LIN {X 0.241,Y -599.129,Z 1375.125,A 0.000,B 0.000,C 90.000,E1 58.408} C_DIS
LIN {X 0.169,Y -600.635,Z 1375.116,A 0.000,B 0.000,C 90.000,E1 56.834} C_DIS
LIN {X -0.271,Y -601.408,Z 1375.111,A 0.000,B 0.000,C 90.000,E1 56.087} C_DIS
LIN {X 0.294,Y -603.031,Z 1375.101,A 0.000,B 0.000,C 90.000,E1 54.196} C_DIS
LIN {X -0.072,Y -604.729,Z 1375.091,A 0.000,B 0.000,C 90.000,E1 52.396} C_DIS
LIN {X -0.082,Y -605.645,Z 1375.084,A 0.000,B 0.000,C 90.000,E1 51.090} C_DIS
LIN {X 0.038,Y -606.172,Z 1375.078,A 0.000,B 0.000,C 90.000,E1 50.033} C_DIS
LIN {X -0.227,Y -606.705,Z 1375.072,A 0.000,B 0.000,C 90.000,E1 49.013} C_DIS
LIN {X -0.356,Y -607.003,Z 1375.068,A 0.000,B 0.000,C 90.000,E1 48.243} C_DIS
LIN {X -0.003,Y -607.306,Z 1375.061,A 0.000,B 0.000,C 90.000,E1 46.905} C_DIS
LIN {X 0.356,Y -607.367,Z 1375.053,A 0.000,B 0.000,C 90.000,E1 45.567} C_DIS
LIN {X -0.205,Y -607.319,Z 1375.049,A 0.000,B 0.000,C 90.000,E1 44.838} C_DIS
LIN {X -0.286,Y -606.975,Z 1375.042,A 0.000,B 0.000,C 90.000,E1 43.542} C_DIS
LIN {X 0.058,Y -606.352,Z 1375.035,A 0.000,B 0.000,C 90.000,E1 42.204} C_DIS
LIN {X -0.017,Y -605.691,Z 1375.027,A 0.000,B 0.000,C 90.000,E1 40.906} C_DIS
LIN {X 0.357,Y -604.817,Z 1375.020,A 0.000,B 0.000,C 90.000,E1 39.564} C_DIS
LIN {X -0.137,Y -603.773,Z 1375.013,A 0.000,B 0.000,C 90.000,E1 38.302} C_DIS
LIN {X -0.179,Y -602.457,Z 1375.005,A 0.000,B 0.000,C 90.000,E1 36.996} C_DIS
LIN {X 0.222,Y -601.485,Z 1375.001,A 0.000,B 0.000,C 90.000,E1 36.171} C_DIS
LIN {X -0.113,Y -599.795,Z 1374.995,A 0.000,B 0.000,C 90.000,E1 35.152} C_DIS
LIN {X -0.215,Y -599.352,Z 1374.994,A 0.000,B 0.000,C 90.000,E1 34.898} C_DIS
LIN {X -0.198,Y -596.501,Z 1374.986,A 0.000,B 0.000,C 90.000,E1 33.579} C_DIS
LIN {X 0.149,Y -594.609,Z 1374.982,A 0.000,B 0.000,C 90.000,E1 32.752} C_DIS
LIN {X -0.345,Y -592.452,Z 1374.978,A 0.000,B 0.000,C 90.000,E1 32.005} C_DIS
LIN {X -0.050,Y -590.090,Z 1374.973,A 0.000,B 0.000,C 90.000,E1 31.180} C_DIS
LIN {X -0.205,Y -586.275,Z 1374.967,A 0.000,B 0.000,C 90.000,E1 30.129} C_DIS
LIN {X 0.229,Y -583.094,Z 1374.963,A 0.000,B 0.000,C 90.000,E1 29.283} C_DIS
LIN {X 0.119,Y -579.414,Z 1374.958,A 0.000,B 0.000,C 90.000,E1 28.487} C_DIS
LIN {X -0.235,Y -576.095,Z 1374.955,A 0.000,B 0.000,C 90.000,E1 27.847} C_DIS
LIN {X 0.082,Y -571.788,Z 1374.950,A 0.000,B 0.000,C 90.000,E1 27.001} C_DIS
LIN {X 0.091,Y -567.040,Z 1374.946,A 0.000,B 0.000,C 90.000,E1 26.181} C_DIS
LIN {X -0.022,Y -563.676,Z 1374.943,A 0.000,B 0.000,C 90.000,E1 25.643} C_DIS
LIN {X -0.098,Y -558.415,Z 1374.938,A 0.000,B 0.000,C 90.000,E1 24.823} C_DIS
LIN {X 0.162,Y -551.372,Z 1374.932,A 0.000,B 0.000,C 90.000,E1 23.823} C_DIS
LIN {X 0.076,Y -545.974,Z 1374.929,A 0.000,B 0.000,C 90.000,E1 23.131} C_DIS
LIN {X -0.265,Y -540.164,Z 1374.925,A 0.000,B 0.000,C 90.000,E1 22.461} C_DIS
LIN {X -0.093,Y -532.857,Z 1374.920,A 0.000,B 0.000,C 90.000,E1 21.589} C_DIS
LIN {X -0.184,Y -522.480,Z 1374.914,A 0.000,B 0.000,C 90.000,E1 20.482} C_DIS
LIN {X -0.189,Y -513.235,Z 1374.908,A 0.000,B 0.000,C 90.000,E1 19.504} C_DIS
LIN {X -0.122,Y -502.645,Z 1374.902,A 0.000,B 0.000,C 90.000,E1 18.417} C_DIS
LIN {X 0.112,Y -491.666,Z 1374.896,A 0.000,B 0.000,C 90.000,E1 17.275} C_DIS
LIN {X -0.037,Y -476.636,Z 1374.888,A 0.000,B 0.000,C 90.000,E1 15.788} C_DIS
LIN {X 0.103,Y -466.836,Z 1374.882,A 0.000,B 0.000,C 90.000,E1 14.773} C_DIS
LIN {X 0.103,Y -454.064,Z 1374.875,A 0.000,B 0.000,C 90.000,E1 13.480} C_DIS
LIN {X -0.045,Y -437.083,Z 1374.865,A 0.000,B 0.000,C 90.000,E1 11.715} C_DIS
LIN {X -0.036,Y -421.953,Z 1374.856,A 0.000,B 0.000,C 90.000,E1 10.018} C_DIS
LIN {X 0.137,Y -410.842,Z 1374.848,A 0.000,B 0.000,C 90.000,E1 8.690} C_DIS
LIN {X 0.106,Y -402.395,Z 1374.843,A 0.000,B 0.000,C 90.000,E1 7.701} C_DIS
LIN {X -0.087,Y -396.749,Z 1374.839,A 0.000,B 0.000,C 90.000,E1 7.068} C_DIS
LIN {X -0.005,Y -393.047,Z 1374.836,A 0.000,B 0.000,C 90.000,E1 6.549} C_DIS
LIN {X -0.180,Y -391.673,Z 1374.835,A 0.000,B 0.000,C 90.000,E1 6.315} C_DIS
LIN {X 0.172,Y -391.657,Z 1374.835,A 0.000,B 0.000,C 90.000,E1 6.258} C_DIS
LIN {X 0.125,Y -394.271,Z 1374.833,A 0.000,B 0.000,C 90.000,E1 5.910} C_DIS
LIN {X 0.119,Y -398.146,Z 1374.831,A 0.000,B 0.000,C 90.000,E1 5.568} C_DIS
LIN {X 0.042,Y -406.599,Z 1374.828,A 0.000,B 0.000,C 90.000,E1 4.935} C_DIS
LIN {X -0.167,Y -411.326,Z 1374.825,A 0.000,B 0.000,C 90.000,E1 4.588} C_DIS
LIN {X -0.196,Y -415.671,Z 1374.823,A 0.000,B 0.000,C 90.000,E1 4.188} C_DIS
LIN {X 0.010,Y -419.888,Z 1374.821,A 0.000,B 0.000,C 90.000,E1 3.726} C_DIS
LIN {X 0.095,Y -424.949,Z 1374.818,A 0.000,B 0.000,C 90.000,E1 3.154} C_DIS
LIN {X -0.129,Y -430.292,Z 1374.814,A 0.000,B 0.000,C 90.000,E1 2.522} C_DIS
LIN {X -0.086,Y -436.249,Z 1374.810,A 0.000,B 0.000,C 90.000,E1 1.718} C_DIS
LIN {X 0.170,Y -442.273,Z 1374.805,A 0.000,B 0.000,C 90.000,E1 0.859} C_DIS
LIN {X 0.000,Y -448.347,Z 1374.800,A 0.000,B 0.000,C 90.000,E1 360.000} C_DIS
LIN {X 0.033,Y -453.864,Z 1374.795,A 0.000,B 0.000,C 90.000,E1 359.141} C_DIS
LIN {X 0.020,Y -458.743,Z 1374.791,A 0.000,B 0.000,C 90.000,E1 358.339} C_DIS
LIN {X -0.035,Y -462.399,Z 1374.787,A 0.000,B 0.000,C 90.000,E1 357.707} C_DIS
LIN {X 0.164,Y -467.432,Z 1374.782,A 0.000,B 0.000,C 90.000,E1 356.731} C_DIS
LIN {X 0.153,Y -470.561,Z 1374.778,A 0.000,B 0.000,C 90.000,E1 356.102} C_DIS
LIN {X -0.152,Y -474.160,Z 1374.774,A 0.000,B 0.000,C 90.000,E1 355.355} C_DIS
LIN {X 0.222,Y -478.076,Z 1374.769,A 0.000,B 0.000,C 90.000,E1 354.375} C_DIS
LIN {X -0.150,Y -480.507,Z 1374.766,A 0.000,B 0.000,C 90.000,E1 353.799} C_DIS
LIN {X -0.181,Y -483.879,Z 1374.760,A 0.000,B 0.000,C 90.000,E1 352.875} C_DIS
LIN {X -0.040,Y -485.914,Z 1374.757,A 0.000,B 0.000,C 90.000,E1 352.243} C_DIS
LIN {X -0.013,Y -488.702,Z 1374.752,A 0.000,B 0.000,C 90.000,E1 351.319} C_DIS
LIN {X -0.250,Y -490.361,Z 1374.748,A 0.000,B 0.000,C 90.000,E1 350.735} C_DIS
LIN {X -0.196,Y -493.358,Z 1374.742,A 0.000,B 0.000,C 90.000,E1 349.511} C_DIS
LIN {X 0.092,Y -494.730,Z 1374.738,A 0.000,B 0.000,C 90.000,E1 348.870} C_DIS
LIN {X -0.002,Y -495.337,Z 1374.737,A 0.000,B 0.000,C 90.000,E1 348.578} C_DIS
LIN {X -0.094,Y -495.813,Z 1374.735,A 0.000,B 0.000,C 90.000,E1 348.285} C_DIS
LIN {X -0.184,Y -496.075,Z 1374.733,A 0.000,B 0.000,C 90.000,E1 347.993} C_DIS
LIN {X 0.212,Y -496.110,Z 1374.732,A 0.000,B 0.000,C 90.000,E1 347.645} C_DIS
LIN {X 0.123,Y -495.824,Z 1374.730,A 0.000,B 0.000,C 90.000,E1 347.353} C_DIS
LIN {X 0.034,Y -494.778,Z 1374.728,A 0.000,B 0.000,C 90.000,E1 347.061} C_DIS
LIN {X -0.129,Y -493.185,Z 1374.727,A 0.000,B 0.000,C 90.000,E1 346.937} C_DIS
LIN {X 0.101,Y -455.532,Z 1374.721,A 0.000,B 0.000,C 90.000,E1 345.825} C_DIS
LIN {X 0.169,Y -423.917,Z 1374.715,A 0.000,B 0.000,C 90.000,E1 344.755} C_DIS
LIN {X 0.093,Y -395.987,Z 1374.709,A 0.000,B 0.000,C 90.000,E1 343.685} C_DIS
LIN {X 0.175,Y -371.706,Z 1374.703,A 0.000,B 0.000,C 90.000,E1 342.598} C_DIS
LIN {X 0.086,Y -360.270,Z 1374.700,A 0.000,B 0.000,C 90.000,E1 342.054} C_DIS
LIN {X 0.052,Y -360.184,Z 1374.700,A 0.000,B 0.000,C 90.000,E1 342.054} C_DIS
LIN {X -0.028,Y -361.934,Z 1374.683,A 0.000,B 0.000,C 90.000,E1 338.954} C_DIS
LIN {X -0.170,Y -366.154,Z 1374.642,A 0.000,B 0.000,C 90.000,E1 331.513} C_DIS
LIN {X 0.050,Y -371.141,Z 1374.605,A 0.000,B 0.000,C 90.000,E1 324.815} C_DIS
LIN {X -0.178,Y -371.570,Z 1374.603,A 0.000,B 0.000,C 90.000,E1 324.482} C_DIS
LIN {X 0.098,Y -372.300,Z 1374.596,A 0.000,B 0.000,C 90.000,E1 323.336} C_DIS
LIN {X 0.155,Y -378.074,Z 1374.564,A 0.000,B 0.000,C 90.000,E1 317.472} C_DIS
LIN {X 0.177,Y -384.183,Z 1374.530,A 0.000,B 0.000,C 90.000,E1 311.310} C_DIS
LIN {X -0.070,Y -384.685,Z 1374.528,A 0.000,B 0.000,C 90.000,E1 310.987} C_DIS
LIN {X -0.170,Y -385.795,Z 1374.520,A 0.000,B 0.000,C 90.000,E1 309.564} C_DIS
LIN {X -0.011,Y -391.319,Z 1374.492,A 0.000,B 0.000,C 90.000,E1 304.532} C_DIS
LIN {X 0.135,Y -397.031,Z 1374.458,A 0.000,B 0.000,C 90.000,E1 298.487} C_DIS
LIN {X -0.084,Y -401.405,Z 1374.427,A 0.000,B 0.000,C 90.000,E1 292.898} C_DIS
LIN {X 0.151,Y -401.668,Z 1374.425,A 0.000,B 0.000,C 90.000,E1 292.514} C_DIS
LIN {X -0.104,Y -404.762,Z 1374.394,A 0.000,B 0.000,C 90.000,E1 286.968} C_DIS
LIN {X -0.209,Y -406.158,Z 1374.363,A 0.000,B 0.000,C 90.000,E1 281.422} C_DIS
LIN {X -0.105,Y -405.652,Z 1374.333,A 0.000,B 0.000,C 90.000,E1 275.853} C_DIS
LIN {X -0.033,Y -403.559,Z 1374.305,A 0.000,B 0.000,C 90.000,E1 270.974} C_DIS
LIN {X -0.098,Y -403.120,Z 1374.302,A 0.000,B 0.000,C 90.000,E1 270.286} C_DIS
LIN {X 0.131,Y -399.041,Z 1374.272,A 0.000,B 0.000,C 90.000,E1 265.008} C_DIS
LIN {X 0.072,Y -398.696,Z 1374.271,A 0.000,B 0.000,C 90.000,E1 264.666} C_DIS
LIN {X -0.046,Y -393.247,Z 1374.243,A 0.000,B 0.000,C 90.000,E1 259.746} C_DIS
LIN {X -0.085,Y -392.976,Z 1374.241,A 0.000,B 0.000,C 90.000,E1 259.398} C_DIS
LIN {X -0.126,Y -392.577,Z 1374.239,A 0.000,B 0.000,C 90.000,E1 259.050} C_DIS
LIN {X 0.033,Y -386.186,Z 1374.213,A 0.000,B 0.000,C 90.000,E1 254.393} C_DIS
LIN {X -0.004,Y -385.081,Z 1374.207,A 0.000,B 0.000,C 90.000,E1 253.323} C_DIS
LIN {X 0.100,Y -378.210,Z 1374.183,A 0.000,B 0.000,C 90.000,E1 248.975} C_DIS
LIN {X -0.044,Y -375.993,Z 1374.173,A 0.000,B 0.000,C 90.000,E1 247.177} C_DIS
LIN {X 0.067,Y -369.190,Z 1374.151,A 0.000,B 0.000,C 90.000,E1 243.127} C_DIS
LIN {X -0.025,Y -366.331,Z 1374.139,A 0.000,B 0.000,C 90.000,E1 240.923} C_DIS
LIN {X 0.133,Y -358.937,Z 1374.114,A 0.000,B 0.000,C 90.000,E1 236.421} C_DIS
LIN {X -0.078,Y -356.112,Z 1374.101,A 0.000,B 0.000,C 90.000,E1 234.196} C_DIS
LIN {X 0.018,Y -349.041,Z 1374.076,A 0.000,B 0.000,C 90.000,E1 229.622} C_DIS
LIN {X -0.016,Y -345.986,Z 1374.061,A 0.000,B 0.000,C 90.000,E1 226.944} C_DIS
LIN {X -0.043,Y -339.190,Z 1374.033,A 0.000,B 0.000,C 90.000,E1 221.919} C_DIS
LIN {X 0.045,Y -337.008,Z 1374.020,A 0.000,B 0.000,C 90.000,E1 219.564} C_DIS
LIN {X 0.021,Y -336.054,Z 1374.016,A 0.000,B 0.000,C 90.000,E1 218.785} C_DIS
LIN {X -0.099,Y -330.416,Z 1373.985,A 0.000,B 0.000,C 90.000,E1 213.293} C_DIS
LIN {X 0.206,Y -329.135,Z 1373.974,A 0.000,B 0.000,C 90.000,E1 211.258} C_DIS
LIN {X 0.083,Y -324.407,Z 1373.938,A 0.000,B 0.000,C 90.000,E1 204.899} C_DIS
LIN {X 0.071,Y -323.717,Z 1373.927,A 0.000,B 0.000,C 90.000,E1 202.898} C_DIS
LIN {X -0.060,Y -322.264,Z 1373.914,A 0.000,B 0.000,C 90.000,E1 200.556} C_DIS
LIN {X -0.078,Y -322.271,Z 1373.914,A 0.000,B 0.000,C 90.000,E1 200.556} C_DIS
LIN {X 0.093,Y -344.041,Z 1373.907,A 0.000,B 0.000,C 90.000,E1 199.214} C_DIS
LIN {X 0.091,Y -367.098,Z 1373.900,A 0.000,B 0.000,C 90.000,E1 198.000} C_DIS
LIN {X -0.130,Y -393.883,Z 1373.893,A 0.000,B 0.000,C 90.000,E1 196.804} C_DIS
LIN {X -0.144,Y -422.596,Z 1373.887,A 0.000,B 0.000,C 90.000,E1 195.662} C_DIS
LIN {X -0.056,Y -440.653,Z 1373.883,A 0.000,B 0.000,C 90.000,E1 195.009} C_DIS
LIN {X -0.145,Y -443.464,Z 1373.883,A 0.000,B 0.000,C 90.000,E1 194.898} C_DIS
LIN {X 0.077,Y -444.638,Z 1373.882,A 0.000,B 0.000,C 90.000,E1 194.717} C_DIS
LIN {X 0.212,Y -445.410,Z 1373.881,A 0.000,B 0.000,C 90.000,E1 194.537} C_DIS
LIN {X -0.084,Y -445.964,Z 1373.880,A 0.000,B 0.000,C 90.000,E1 194.411} C_DIS
LIN {X 0.082,Y -446.725,Z 1373.878,A 0.000,B 0.000,C 90.000,E1 194.064} C_DIS
LIN {X -0.182,Y -447.189,Z 1373.876,A 0.000,B 0.000,C 90.000,E1 193.772} C_DIS
LIN {X 0.098,Y -447.488,Z 1373.875,A 0.000,B 0.000,C 90.000,E1 193.411} C_DIS
LIN {X 0.044,Y -447.972,Z 1373.867,A 0.000,B 0.000,C 90.000,E1 192.119} C_DIS
LIN {X -0.092,Y -448.344,Z 1373.860,A 0.000,B 0.000,C 90.000,E1 190.838} C_DIS
LIN {X -0.031,Y -448.520,Z 1373.851,A 0.000,B 0.000,C 90.000,E1 189.208} C_DIS
LIN {X -0.108,Y -448.510,Z 1373.839,A 0.000,B 0.000,C 90.000,E1 186.947} C_DIS
LIN {X 0.087,Y -448.469,Z 1373.831,A 0.000,B 0.000,C 90.000,E1 185.625} C_DIS
LIN {X 0.145,Y -448.331,Z 1373.826,A 0.000,B 0.000,C 90.000,E1 184.645} C_DIS
LIN {X -0.140,Y -447.861,Z 1373.819,A 0.000,B 0.000,C 90.000,E1 183.383} C_DIS
LIN {X 0.176,Y -447.483,Z 1373.815,A 0.000,B 0.000,C 90.000,E1 182.694} C_DIS
LIN {X 0.181,Y -446.518,Z 1373.810,A 0.000,B 0.000,C 90.000,E1 181.718} C_DIS
LIN {X 0.020,Y -445.840,Z 1373.806,A 0.000,B 0.000,C 90.000,E1 181.088} C_DIS
LIN {X -0.143,Y -445.025,Z 1373.802,A 0.000,B 0.000,C 90.000,E1 180.458} C_DIS
LIN {X -0.176,Y -443.449,Z 1373.797,A 0.000,B 0.000,C 90.000,E1 179.484} C_DIS
LIN {X 0.086,Y -442.211,Z 1373.793,A 0.000,B 0.000,C 90.000,E1 178.797} C_DIS
LIN {X 0.029,Y -439.643,Z 1373.788,A 0.000,B 0.000,C 90.000,E1 177.822} C_DIS
LIN {X -0.181,Y -437.692,Z 1373.784,A 0.000,B 0.000,C 90.000,E1 177.192} C_DIS
LIN {X 0.053,Y -435.361,Z 1373.781,A 0.000,B 0.000,C 90.000,E1 176.502} C_DIS
LIN {X 0.192,Y -433.388,Z 1373.778,A 0.000,B 0.000,C 90.000,E1 175.988} C_DIS
LIN {X -0.047,Y -430.543,Z 1373.774,A 0.000,B 0.000,C 90.000,E1 175.355} C_DIS
LIN {X 0.216,Y -425.262,Z 1373.769,A 0.000,B 0.000,C 90.000,E1 174.318} C_DIS
LIN {X -0.006,Y -418.909,Z 1373.763,A 0.000,B 0.000,C 90.000,E1 173.337} C_DIS
LIN {X 0.112,Y -412.069,Z 1373.757,A 0.000,B 0.000,C 90.000,E1 172.299} C_DIS
LIN {X 0.155,Y -398.379,Z 1373.746,A 0.000,B 0.000,C 90.000,E1 170.218} C_DIS
LIN {X 0.055,Y -387.770,Z 1373.736,A 0.000,B 0.000,C 90.000,E1 168.465} C_DIS
LIN {X -0.070,Y -383.203,Z 1373.731,A 0.000,B 0.000,C 90.000,E1 167.589} C_DIS
LIN {X 0.044,Y -380.586,Z 1373.727,A 0.000,B 0.000,C 90.000,E1 166.881} C_DIS
LIN {X 0.042,Y -380.052,Z 1373.726,A 0.000,B 0.000,C 90.000,E1 166.700} C_DIS
LIN {X -0.148,Y -380.021,Z 1373.724,A 0.000,B 0.000,C 90.000,E1 166.353} C_DIS
LIN {X -0.169,Y -380.030,Z 1373.724,A 0.000,B 0.000,C 90.000,E1 166.353} C_DIS
LIN {X -0.062,Y -381.121,Z 1373.723,A 0.000,B 0.000,C 90.000,E1 166.117} C_DIS
LIN {X -0.050,Y -382.411,Z 1373.721,A 0.000,B 0.000,C 90.000,E1 165.811} C_DIS
LIN {X 0.017,Y -387.298,Z 1373.718,A 0.000,B 0.000,C 90.000,E1 165.172} C_DIS
LIN {X -0.039,Y -393.789,Z 1373.714,A 0.000,B 0.000,C 90.000,E1 164.448} C_DIS
LIN {X -0.086,Y -400.930,Z 1373.710,A 0.000,B 0.000,C 90.000,E1 163.740} C_DIS
LIN {X 0.039,Y -416.462,Z 1373.702,A 0.000,B 0.000,C 90.000,E1 162.308} C_DIS
LIN {X 0.224,Y -441.867,Z 1373.690,A 0.000,B 0.000,C 90.000,E1 160.242} C_DIS
LIN {X -0.082,Y -454.491,Z 1373.685,A 0.000,B 0.000,C 90.000,E1 159.316} C_DIS
LIN {X -0.007,Y -460.608,Z 1373.682,A 0.000,B 0.000,C 90.000,E1 158.827} C_DIS
LIN {X -0.071,Y -468.194,Z 1373.679,A 0.000,B 0.000,C 90.000,E1 158.209} C_DIS
LIN {X 0.167,Y -475.655,Z 1373.675,A 0.000,B 0.000,C 90.000,E1 157.539} C_DIS
LIN {X -0.219,Y -484.360,Z 1373.671,A 0.000,B 0.000,C 90.000,E1 156.794} C_DIS
LIN {X -0.096,Y -492.955,Z 1373.667,A 0.000,B 0.000,C 90.000,E1 155.973} C_DIS
LIN {X -0.149,Y -501.060,Z 1373.662,A 0.000,B 0.000,C 90.000,E1 155.153} C_DIS
LIN {X -0.035,Y -505.036,Z 1373.660,A 0.000,B 0.000,C 90.000,E1 154.717} C_DIS
LIN {X 0.113,Y -511.378,Z 1373.656,A 0.000,B 0.000,C 90.000,E1 153.973} C_DIS
LIN {X -0.074,Y -517.595,Z 1373.651,A 0.000,B 0.000,C 90.000,E1 153.256} C_DIS
LIN {X 0.254,Y -523.274,Z 1373.647,A 0.000,B 0.000,C 90.000,E1 152.487} C_DIS
LIN {X -0.227,Y -526.484,Z 1373.645,A 0.000,B 0.000,C 90.000,E1 152.103} C_DIS
LIN {X -0.133,Y -530.224,Z 1373.642,A 0.000,B 0.000,C 90.000,E1 151.513} C_DIS
LIN {X -0.156,Y -534.214,Z 1373.638,A 0.000,B 0.000,C 90.000,E1 150.795} C_DIS
LIN {X -0.002,Y -536.963,Z 1373.635,A 0.000,B 0.000,C 90.000,E1 150.205} C_DIS
LIN {X 0.165,Y -540.360,Z 1373.630,A 0.000,B 0.000,C 90.000,E1 149.331} C_DIS
LIN {X -0.103,Y -542.398,Z 1373.627,A 0.000,B 0.000,C 90.000,E1 148.791} C_DIS
LIN {X 0.106,Y -544.198,Z 1373.623,A 0.000,B 0.000,C 90.000,E1 148.201} C_DIS
LIN {X -0.107,Y -546.401,Z 1373.619,A 0.000,B 0.000,C 90.000,E1 147.375} C_DIS
LIN {X 0.125,Y -547.666,Z 1373.616,A 0.000,B 0.000,C 90.000,E1 146.786} C_DIS
LIN {X -0.052,Y -549.270,Z 1373.611,A 0.000,B 0.000,C 90.000,E1 145.960} C_DIS
LIN {X 0.157,Y -551.091,Z 1373.605,A 0.000,B 0.000,C 90.000,E1 144.815} C_DIS
LIN {X 0.014,Y -552.233,Z 1373.600,A 0.000,B 0.000,C 90.000,E1 143.989} C_DIS
LIN {X 0.273,Y -553.255,Z 1373.594,A 0.000,B 0.000,C 90.000,E1 142.844} C_DIS
LIN {X 0.181,Y -554.267,Z 1373.586,A 0.000,B 0.000,C 90.000,E1 141.457} C_DIS
LIN {X 0.033,Y -555.029,Z 1373.580,A 0.000,B 0.000,C 90.000,E1 140.356} C_DIS
LIN {X 0.320,Y -555.830,Z 1373.572,A 0.000,B 0.000,C 90.000,E1 138.933} C_DIS
LIN {X 0.200,Y -556.587,Z 1373.564,A 0.000,B 0.000,C 90.000,E1 137.553} C_DIS
LIN {X -0.318,Y -557.169,Z 1373.557,A 0.000,B 0.000,C 90.000,E1 136.215} C_DIS
LIN {X 0.014,Y -557.779,Z 1373.547,A 0.000,B 0.000,C 90.000,E1 134.514} C_DIS
LIN {X -0.099,Y -558.296,Z 1373.540,A 0.000,B 0.000,C 90.000,E1 133.137} C_DIS
LIN {X -0.180,Y -558.783,Z 1373.532,A 0.000,B 0.000,C 90.000,E1 131.757} C_DIS
LIN {X 0.011,Y -559.850,Z 1373.520,A 0.000,B 0.000,C 90.000,E1 129.519} C_DIS
LIN {X -0.046,Y -560.355,Z 1373.517,A 0.000,B 0.000,C 90.000,E1 129.116} C_DIS
LIN {X -0.082,Y -561.346,Z 1373.515,A 0.000,B 0.000,C 90.000,E1 128.705} C_DIS
LIN {X 0.082,Y -561.467,Z 1373.515,A 0.000,B 0.000,C 90.000,E1 128.588} C_DIS
LIN {X 0.040,Y -561.486,Z 1373.514,A 0.000,B 0.000,C 90.000,E1 128.588} C_DIS
LIN {X -0.088,Y -562.514,Z 1373.514,A 0.000,B 0.000,C 90.000,E1 128.463} C_DIS
LIN {X -0.117,Y -564.716,Z 1373.513,A 0.000,B 0.000,C 90.000,E1 128.338} C_DIS
LIN {X -0.017,Y -569.709,Z 1373.512,A 0.000,B 0.000,C 90.000,E1 128.177} C_DIS
LIN {X 0.216,Y -572.168,Z 1373.512,A 0.000,B 0.000,C 90.000,E1 128.096} C_DIS
LIN {X -0.017,Y -578.338,Z 1373.511,A 0.000,B 0.000,C 90.000,E1 127.935} C_DIS
LIN {X 0.144,Y -581.541,Z 1373.510,A 0.000,B 0.000,C 90.000,E1 127.810} C_DIS
LIN {X -0.252,Y -584.383,Z 1373.510,A 0.000,B 0.000,C 90.000,E1 127.729} C_DIS
LIN {X -0.065,Y -587.357,Z 1373.509,A 0.000,B 0.000,C 90.000,E1 127.569} C_DIS
LIN {X 0.067,Y -590.363,Z 1373.508,A 0.000,B 0.000,C 90.000,E1 127.397} C_DIS
LIN {X -0.042,Y -593.196,Z 1373.507,A 0.000,B 0.000,C 90.000,E1 127.237} C_DIS
LIN {X -0.077,Y -598.802,Z 1373.505,A 0.000,B 0.000,C 90.000,E1 126.870} C_DIS
LIN {X -0.088,Y -604.276,Z 1373.503,A 0.000,B 0.000,C 90.000,E1 126.457} C_DIS
LIN {X 0.234,Y -608.428,Z 1373.501,A 0.000,B 0.000,C 90.000,E1 126.091} C_DIS
LIN {X 0.068,Y -614.929,Z 1373.497,A 0.000,B 0.000,C 90.000,E1 125.518} C_DIS
LIN {X 0.120,Y -621.206,Z 1373.494,A 0.000,B 0.000,C 90.000,E1 124.898} C_DIS
LIN {X 0.012,Y -626.001,Z 1373.491,A 0.000,B 0.000,C 90.000,E1 124.405} C_DIS
LIN {X -0.152,Y -630.526,Z 1373.488,A 0.000,B 0.000,C 90.000,E1 123.913} C_DIS
LIN {X -0.295,Y -636.832,Z 1373.484,A 0.000,B 0.000,C 90.000,E1 123.166} C_DIS
LIN {X 0.142,Y -641.613,Z 1373.481,A 0.000,B 0.000,C 90.000,E1 122.498} C_DIS
LIN {X 0.082,Y -646.017,Z 1373.477,A 0.000,B 0.000,C 90.000,E1 121.878} C_DIS
LIN {X 0.013,Y -649.279,Z 1373.474,A 0.000,B 0.000,C 90.000,E1 121.386} C_DIS
LIN {X 0.183,Y -652.248,Z 1373.472,A 0.000,B 0.000,C 90.000,E1 120.875} C_DIS
LIN {X 0.332,Y -655.444,Z 1373.468,A 0.000,B 0.000,C 90.000,E1 120.256} C_DIS
LIN {X 0.093,Y -658.704,Z 1373.464,A 0.000,B 0.000,C 90.000,E1 119.539} C_DIS
LIN {X -0.113,Y -661.218,Z 1373.460,A 0.000,B 0.000,C 90.000,E1 118.821} C_DIS
LIN {X -0.294,Y -662.986,Z 1373.456,A 0.000,B 0.000,C 90.000,E1 118.103} C_DIS
LIN {X -0.013,Y -663.616,Z 1373.453,A 0.000,B 0.000,C 90.000,E1 117.590} C_DIS
LIN {X -0.172,Y -663.947,Z 1373.449,A 0.000,B 0.000,C 90.000,E1 116.873} C_DIS
LIN {X 0.261,Y -663.727,Z 1373.445,A 0.000,B 0.000,C 90.000,E1 116.104} C_DIS
LIN {X -0.194,Y -663.079,Z 1373.441,A 0.000,B 0.000,C 90.000,E1 115.412} C_DIS
LIN {X 0.090,Y -662.419,Z 1373.438,A 0.000,B 0.000,C 90.000,E1 114.899} C_DIS
LIN {X 0.364,Y -661.332,Z 1373.436,A 0.000,B 0.000,C 90.000,E1 114.387} C_DIS
LIN {X -0.308,Y -659.518,Z 1373.434,A 0.000,B 0.000,C 90.000,E1 114.079} C_DIS
LIN {X -0.179,Y -658.193,Z 1373.432,A 0.000,B 0.000,C 90.000,E1 113.823} C_DIS
LIN {X -0.116,Y -657.327,Z 1373.432,A 0.000,B 0.000,C 90.000,E1 113.695} C_DIS
LIN {X 0.020,Y -652.195,Z 1373.429,A 0.000,B 0.000,C 90.000,E1 113.206} C_DIS
LIN {X 0.139,Y -650.458,Z 1373.428,A 0.000,B 0.000,C 90.000,E1 113.078} C_DIS
LIN {X -0.075,Y -641.037,Z 1373.426,A 0.000,B 0.000,C 90.000,E1 112.695} C_DIS
LIN {X -0.275,Y -638.847,Z 1373.426,A 0.000,B 0.000,C 90.000,E1 112.642} C_DIS
LIN {X -0.164,Y -625.698,Z 1373.424,A 0.000,B 0.000,C 90.000,E1 112.280} C_DIS
LIN {X 0.113,Y -624.079,Z 1373.423,A 0.000,B 0.000,C 90.000,E1 112.206} C_DIS
LIN {X 0.063,Y -623.937,Z 1373.423,A 0.000,B 0.000,C 90.000,E1 112.206} C_DIS
LIN {X 0.015,Y -633.461,Z 1373.418,A 0.000,B 0.000,C 90.000,E1 111.173} C_DIS
LIN {X 0.068,Y -637.802,Z 1373.415,A 0.000,B 0.000,C 90.000,E1 110.663} C_DIS
LIN {X -0.279,Y -642.498,Z 1373.411,A 0.000,B 0.000,C 90.000,E1 110.066} C_DIS
LIN {X 0.270,Y -647.230,Z 1373.407,A 0.000,B 0.000,C 90.000,E1 109.268} C_DIS
LIN {X 0.006,Y -650.612,Z 1373.404,A 0.000,B 0.000,C 90.000,E1 108.671} C_DIS
LIN {X -0.114,Y -655.501,Z 1373.398,A 0.000,B 0.000,C 90.000,E1 107.692} C_DIS
LIN {X 0.354,Y -658.842,Z 1373.394,A 0.000,B 0.000,C 90.000,E1 106.913} C_DIS
LIN {X 0.138,Y -660.755,Z 1373.391,A 0.000,B 0.000,C 90.000,E1 106.441} C_DIS
LIN {X 0.023,Y -663.168,Z 1373.387,A 0.000,B 0.000,C 90.000,E1 105.717} C_DIS
LIN {X -0.251,Y -664.909,Z 1373.383,A 0.000,B 0.000,C 90.000,E1 105.009} C_DIS
LIN {X 0.222,Y -665.866,Z 1373.381,A 0.000,B 0.000,C 90.000,E1 104.481} C_DIS
LIN {X -0.019,Y -666.847,Z 1373.377,A 0.000,B 0.000,C 90.000,E1 103.772} C_DIS
LIN {X -0.176,Y -667.289,Z 1373.374,A 0.000,B 0.000,C 90.000,E1 103.300} C_DIS
LIN {X -0.330,Y -667.473,Z 1373.371,A 0.000,B 0.000,C 90.000,E1 102.827} C_DIS
LIN {X 0.090,Y -667.413,Z 1373.367,A 0.000,B 0.000,C 90.000,E1 102.063} C_DIS
LIN {X -0.068,Y -667.171,Z 1373.364,A 0.000,B 0.000,C 90.000,E1 101.591} C_DIS
LIN {X -0.359,Y -666.661,Z 1373.362,A 0.000,B 0.000,C 90.000,E1 101.130} C_DIS
LIN {X 0.045,Y -665.509,Z 1373.358,A 0.000,B 0.000,C 90.000,E1 100.366} C_DIS
LIN {X -0.248,Y -664.512,Z 1373.355,A 0.000,B 0.000,C 90.000,E1 99.905} C_DIS
LIN {X 0.017,Y -662.579,Z 1373.351,A 0.000,B 0.000,C 90.000,E1 99.151} C_DIS
LIN {X -0.081,Y -661.865,Z 1373.349,A 0.000,B 0.000,C 90.000,E1 98.916} C_DIS
LIN {X 0.154,Y -659.278,Z 1373.345,A 0.000,B 0.000,C 90.000,E1 98.163} C_DIS
LIN {X -0.168,Y -657.343,Z 1373.343,A 0.000,B 0.000,C 90.000,E1 97.701} C_DIS
LIN {X 0.020,Y -653.999,Z 1373.339,A 0.000,B 0.000,C 90.000,E1 96.947} C_DIS
LIN {X -0.301,Y -652.112,Z 1373.337,A 0.000,B 0.000,C 90.000,E1 96.606} C_DIS
LIN {X -0.061,Y -648.684,Z 1373.333,A 0.000,B 0.000,C 90.000,E1 95.967} C_DIS
LIN {X -0.042,Y -644.197,Z 1373.329,A 0.000,B 0.000,C 90.000,E1 95.220} C_DIS
LIN {X -0.065,Y -639.450,Z 1373.325,A 0.000,B 0.000,C 90.000,E1 94.473} C_DIS
LIN {X 0.121,Y -635.990,Z 1373.322,A 0.000,B 0.000,C 90.000,E1 93.955} C_DIS
LIN {X 0.239,Y -632.120,Z 1373.319,A 0.000,B 0.000,C 90.000,E1 93.440} C_DIS
LIN {X 0.228,Y -626.450,Z 1373.316,A 0.000,B 0.000,C 90.000,E1 92.808} C_DIS
LIN {X -0.307,Y -618.992,Z 1373.312,A 0.000,B 0.000,C 90.000,E1 92.121} C_DIS
LIN {X -0.041,Y -613.736,Z 1373.309,A 0.000,B 0.000,C 90.000,E1 91.604} C_DIS
LIN {X -0.211,Y -609.783,Z 1373.307,A 0.000,B 0.000,C 90.000,E1 91.260} C_DIS
LIN {X -0.269,Y -603.894,Z 1373.304,A 0.000,B 0.000,C 90.000,E1 90.802} C_DIS
LIN {X 0.072,Y -599.289,Z 1373.303,A 0.000,B 0.000,C 90.000,E1 90.458} C_DIS
LIN {X -0.079,Y -596.205,Z 1373.302,A 0.000,B 0.000,C 90.000,E1 90.286} C_DIS
LIN {X -0.111,Y -589.448,Z 1373.300,A 0.000,B 0.000,C 90.000,E1 89.943} C_DIS
LIN {X 0.164,Y -580.927,Z 1373.298,A 0.000,B 0.000,C 90.000,E1 89.542} C_DIS
LIN {X 0.157,Y -577.475,Z 1373.297,A 0.000,B 0.000,C 90.000,E1 89.370} C_DIS
LIN {X -0.023,Y -574.910,Z 1373.295,A 0.000,B 0.000,C 90.000,E1 89.141} C_DIS
LIN {X -0.151,Y -574.108,Z 1373.295,A 0.000,B 0.000,C 90.000,E1 89.083} C_DIS
LIN {X -0.193,Y -574.081,Z 1373.295,A 0.000,B 0.000,C 90.000,E1 89.083} C_DIS
LIN {X -0.054,Y -573.568,Z 1373.293,A 0.000,B 0.000,C 90.000,E1 88.740} C_DIS
LIN {X -0.114,Y -573.923,Z 1373.289,A 0.000,B 0.000,C 90.000,E1 88.051} C_DIS
LIN {X -0.045,Y -575.752,Z 1373.277,A 0.000,B 0.000,C 90.000,E1 85.869} C_DIS
LIN {X -0.118,Y -578.638,Z 1373.262,A 0.000,B 0.000,C 90.000,E1 83.166} C_DIS
LIN {X 0.100,Y -580.887,Z 1373.251,A 0.000,B 0.000,C 90.000,E1 81.254} C_DIS
LIN {X -0.095,Y -582.490,Z 1373.244,A 0.000,B 0.000,C 90.000,E1 79.926} C_DIS
LIN {X 0.273,Y -583.673,Z 1373.238,A 0.000,B 0.000,C 90.000,E1 78.814} C_DIS
LIN {X 0.092,Y -584.750,Z 1373.232,A 0.000,B 0.000,C 90.000,E1 77.757} C_DIS
LIN {X -0.073,Y -585.709,Z 1373.226,A 0.000,B 0.000,C 90.000,E1 76.700} C_DIS
LIN {X -0.158,Y -586.937,Z 1373.217,A 0.000,B 0.000,C 90.000,E1 75.102} C_DIS
LIN {X 0.095,Y -587.830,Z 1373.210,A 0.000,B 0.000,C 90.000,E1 73.740} C_DIS
LIN {X 0.202,Y -588.849,Z 1373.201,A 0.000,B 0.000,C 90.000,E1 72.127} C_DIS
LIN {X -0.155,Y -589.414,Z 1373.195,A 0.000,B 0.000,C 90.000,E1 71.094} C_DIS
LIN {X 0.038,Y -590.483,Z 1373.185,A 0.000,B 0.000,C 90.000,E1 69.209} C_DIS
LIN {X -0.090,Y -591.611,Z 1373.174,A 0.000,B 0.000,C 90.000,E1 67.358} C_DIS
LIN {X 0.140,Y -592.823,Z 1373.165,A 0.000,B 0.000,C 90.000,E1 65.741} C_DIS
LIN {X -0.249,Y -593.756,Z 1373.159,A 0.000,B 0.000,C 90.000,E1 64.717} C_DIS
LIN {X 0.171,Y -595.179,Z 1373.149,A 0.000,B 0.000,C 90.000,E1 62.820} C_DIS
LIN {X 0.031,Y -596.903,Z 1373.137,A 0.000,B 0.000,C 90.000,E1 60.717} C_DIS
LIN {X 0.029,Y -598.677,Z 1373.127,A 0.000,B 0.000,C 90.000,E1 58.869} C_DIS
LIN {X -0.137,Y -600.435,Z 1373.117,A 0.000,B 0.000,C 90.000,E1 57.041} C_DIS
LIN {X 0.162,Y -601.419,Z 1373.111,A 0.000,B 0.000,C 90.000,E1 55.960} C_DIS
LIN {X 0.234,Y -603.070,Z 1373.101,A 0.000,B 0.000,C 90.000,E1 54.116} C_DIS
LIN {X 0.091,Y -604.524,Z 1373.092,A 0.000,B 0.000,C 90.000,E1 52.557} C_DIS
LIN {X 0.074,Y -605.490,Z 1373.085,A 0.000,B 0.000,C 90.000,E1 51.251} C_DIS
LIN {X 0.189,Y -606.083,Z 1373.079,A 0.000,B 0.000,C 90.000,E1 50.194} C_DIS
LIN {X -0.277,Y -606.722,Z 1373.072,A 0.000,B 0.000,C 90.000,E1 48.933} C_DIS
LIN {X -0.147,Y -607.082,Z 1373.066,A 0.000,B 0.000,C 90.000,E1 47.877} C_DIS
LIN {X 0.202,Y -607.329,Z 1373.059,A 0.000,B 0.000,C 90.000,E1 46.539} C_DIS
LIN {X -0.066,Y -607.362,Z 1373.050,A 0.000,B 0.000,C 90.000,E1 45.000} C_DIS
LIN {X -0.146,Y -607.021,Z 1373.043,A 0.000,B 0.000,C 90.000,E1 43.704} C_DIS
LIN {X 0.394,Y -606.584,Z 1373.037,A 0.000,B 0.000,C 90.000,E1 42.609} C_DIS
LIN {X 0.130,Y -605.772,Z 1373.028,A 0.000,B 0.000,C 90.000,E1 41.067} C_DIS
LIN {X 0.043,Y -604.981,Z 1373.021,A 0.000,B 0.000,C 90.000,E1 39.769} C_DIS
LIN {X 0.280,Y -603.720,Z 1373.012,A 0.000,B 0.000,C 90.000,E1 38.177} C_DIS
LIN {X 0.242,Y -602.416,Z 1373.005,A 0.000,B 0.000,C 90.000,E1 36.870} C_DIS
LIN {X 0.160,Y -601.416,Z 1373.001,A 0.000,B 0.000,C 90.000,E1 36.091} C_DIS
LIN {X 0.067,Y -600.164,Z 1372.996,A 0.000,B 0.000,C 90.000,E1 35.311} C_DIS
LIN {X -0.280,Y -599.249,Z 1372.993,A 0.000,B 0.000,C 90.000,E1 34.818} C_DIS
LIN {X -0.270,Y -596.391,Z 1372.986,A 0.000,B 0.000,C 90.000,E1 33.499} C_DIS
LIN {X 0.075,Y -594.488,Z 1372.982,A 0.000,B 0.000,C 90.000,E1 32.673} C_DIS
LIN {X 0.080,Y -592.307,Z 1372.977,A 0.000,B 0.000,C 90.000,E1 31.878} C_DIS
LIN {X 0.069,Y -589.929,Z 1372.973,A 0.000,B 0.000,C 90.000,E1 31.082} C_DIS
LIN {X 0.214,Y -586.051,Z 1372.967,A 0.000,B 0.000,C 90.000,E1 30.001} C_DIS
LIN {X 0.136,Y -582.824,Z 1372.962,A 0.000,B 0.000,C 90.000,E1 29.205} C_DIS
LIN {X 0.021,Y -579.131,Z 1372.958,A 0.000,B 0.000,C 90.000,E1 28.409} C_DIS
LIN {X 0.246,Y -576.470,Z 1372.955,A 0.000,B 0.000,C 90.000,E1 27.847} C_DIS
LIN {X 0.053,Y -572.188,Z 1372.950,A 0.000,B 0.000,C 90.000,E1 27.052} C_DIS
LIN {X 0.064,Y -567.487,Z 1372.946,A 0.000,B 0.000,C 90.000,E1 26.232} C_DIS
LIN {X 0.217,Y -564.150,Z 1372.943,A 0.000,B 0.000,C 90.000,E1 25.668} C_DIS
LIN {X 0.150,Y -558.862,Z 1372.938,A 0.000,B 0.000,C 90.000,E1 24.847} C_DIS
LIN {X 0.027,Y -552.902,Z 1372.934,A 0.000,B 0.000,C 90.000,E1 24.027} C_DIS
LIN {X 0.079,Y -548.705,Z 1372.930,A 0.000,B 0.000,C 90.000,E1 23.462} C_DIS
LIN {X 0.099,Y -544.253,Z 1372.927,A 0.000,B 0.000,C 90.000,E1 22.898} C_DIS
LIN {X -0.050,Y -538.357,Z 1372.923,A 0.000,B 0.000,C 90.000,E1 22.206} C_DIS
LIN {X -0.108,Y -533.460,Z 1372.920,A 0.000,B 0.000,C 90.000,E1 21.642} C_DIS
LIN {X 0.065,Y -521.682,Z 1372.913,A 0.000,B 0.000,C 90.000,E1 20.355} C_DIS
LIN {X 0.130,Y -512.613,Z 1372.908,A 0.000,B 0.000,C 90.000,E1 19.396} C_DIS
LIN {X -0.032,Y -501.810,Z 1372.902,A 0.000,B 0.000,C 90.000,E1 18.308} C_DIS
LIN {X 0.079,Y -492.541,Z 1372.896,A 0.000,B 0.000,C 90.000,E1 17.347} C_DIS
LIN {X 0.098,Y -477.426,Z 1372.888,A 0.000,B 0.000,C 90.000,E1 15.843} C_DIS
LIN {X 0.039,Y -466.268,Z 1372.882,A 0.000,B 0.000,C 90.000,E1 14.717} C_DIS
LIN {X 0.185,Y -453.506,Z 1372.875,A 0.000,B 0.000,C 90.000,E1 13.411} C_DIS
LIN {X -0.185,Y -437.926,Z 1372.866,A 0.000,B 0.000,C 90.000,E1 11.827} C_DIS
LIN {X 0.142,Y -422.663,Z 1372.856,A 0.000,B 0.000,C 90.000,E1 10.084} C_DIS
LIN {X 0.175,Y -411.711,Z 1372.849,A 0.000,B 0.000,C 90.000,E1 8.803} C_DIS
LIN {X 0.167,Y -401.807,Z 1372.843,A 0.000,B 0.000,C 90.000,E1 7.644} C_DIS
LIN {X -0.052,Y -397.520,Z 1372.840,A 0.000,B 0.000,C 90.000,E1 7.182} C_DIS
LIN {X 0.040,Y -392.562,Z 1372.836,A 0.000,B 0.000,C 90.000,E1 6.486} C_DIS
LIN {X 0.120,Y -391.932,Z 1372.835,A 0.000,B 0.000,C 90.000,E1 6.315} C_DIS
LIN {X 0.084,Y -391.919,Z 1372.835,A 0.000,B 0.000,C 90.000,E1 6.315} C_DIS
LIN {X 0.051,Y -394.002,Z 1372.834,A 0.000,B 0.000,C 90.000,E1 6.030} C_DIS
LIN {X 0.082,Y -397.812,Z 1372.832,A 0.000,B 0.000,C 90.000,E1 5.682} C_DIS
LIN {X -0.154,Y -405.165,Z 1372.829,A 0.000,B 0.000,C 90.000,E1 5.163} C_DIS
LIN {X -0.035,Y -411.431,Z 1372.826,A 0.000,B 0.000,C 90.000,E1 4.645} C_DIS
LIN {X 0.010,Y -415.886,Z 1372.824,A 0.000,B 0.000,C 90.000,E1 4.245} C_DIS
LIN {X 0.012,Y -421.511,Z 1372.820,A 0.000,B 0.000,C 90.000,E1 3.669} C_DIS
LIN {X -0.002,Y -425.601,Z 1372.818,A 0.000,B 0.000,C 90.000,E1 3.212} C_DIS
LIN {X -0.197,Y -429.670,Z 1372.815,A 0.000,B 0.000,C 90.000,E1 2.751} C_DIS
LIN {X 0.088,Y -437.224,Z 1372.810,A 0.000,B 0.000,C 90.000,E1 1.718} C_DIS
LIN {X -0.013,Y -443.246,Z 1372.805,A 0.000,B 0.000,C 90.000,E1 0.917} C_DIS
LIN {X 0.000,Y -449.603,Z 1372.800,A 0.000,B 0.000,C 90.000,E1 360.000} C_DIS
LIN {X 0.044,Y -455.152,Z 1372.795,A 0.000,B 0.000,C 90.000,E1 359.141} C_DIS
LIN {X -0.053,Y -459.122,Z 1372.792,A 0.000,B 0.000,C 90.000,E1 358.511} C_DIS
LIN {X -0.003,Y -463.692,Z 1372.787,A 0.000,B 0.000,C 90.000,E1 357.707} C_DIS
LIN {X 0.073,Y -467.963,Z 1372.783,A 0.000,B 0.000,C 90.000,E1 356.906} C_DIS
LIN {X 0.213,Y -471.907,Z 1372.779,A 0.000,B 0.000,C 90.000,E1 356.102} C_DIS
LIN {X -0.080,Y -475.494,Z 1372.774,A 0.000,B 0.000,C 90.000,E1 355.355} C_DIS
LIN {X 0.133,Y -478.801,Z 1372.770,A 0.000,B 0.000,C 90.000,E1 354.552} C_DIS
LIN {X 0.104,Y -480.696,Z 1372.767,A 0.000,B 0.000,C 90.000,E1 354.090} C_DIS
LIN {X 0.076,Y -484.140,Z 1372.762,A 0.000,B 0.000,C 90.000,E1 353.166} C_DIS
LIN {X -0.264,Y -486.297,Z 1372.759,A 0.000,B 0.000,C 90.000,E1 352.591} C_DIS
LIN {X -0.163,Y -489.134,Z 1372.754,A 0.000,B 0.000,C 90.000,E1 351.659} C_DIS
LIN {X 0.014,Y -490.871,Z 1372.750,A 0.000,B 0.000,C 90.000,E1 351.027} C_DIS
LIN {X 0.176,Y -493.169,Z 1372.745,A 0.000,B 0.000,C 90.000,E1 350.095} C_DIS
LIN {X -0.118,Y -495.384,Z 1372.740,A 0.000,B 0.000,C 90.000,E1 349.218} C_DIS
LIN {X 0.100,Y -497.281,Z 1372.735,A 0.000,B 0.000,C 90.000,E1 348.285} C_DIS
LIN {X -0.068,Y -498.281,Z 1372.732,A 0.000,B 0.000,C 90.000,E1 347.701} C_DIS
LIN {X -0.151,Y -498.579,Z 1372.730,A 0.000,B 0.000,C 90.000,E1 347.409} C_DIS
LIN {X -0.232,Y -498.667,Z 1372.728,A 0.000,B 0.000,C 90.000,E1 347.117} C_DIS
LIN {X 0.173,Y -498.499,Z 1372.727,A 0.000,B 0.000,C 90.000,E1 346.769} C_DIS
LIN {X 0.208,Y -497.839,Z 1372.725,A 0.000,B 0.000,C 90.000,E1 346.464} C_DIS
LIN {X -0.133,Y -497.079,Z 1372.724,A 0.000,B 0.000,C 90.000,E1 346.353} C_DIS
LIN {X 0.126,Y -494.426,Z 1372.723,A 0.000,B 0.000,C 90.000,E1 346.172} C_DIS
LIN {X 0.168,Y -459.639,Z 1372.718,A 0.000,B 0.000,C 90.000,E1 345.117} C_DIS
LIN {X 0.045,Y -428.125,Z 1372.711,A 0.000,B 0.000,C 90.000,E1 344.031} C_DIS
LIN {X 0.086,Y -400.296,Z 1372.705,A 0.000,B 0.000,C 90.000,E1 342.906} C_DIS
LIN {X -0.074,Y -376.115,Z 1372.699,A 0.000,B 0.000,C 90.000,E1 341.819} C_DIS
LIN {X -0.142,Y -360.659,Z 1372.695,A 0.000,B 0.000,C 90.000,E1 341.040} C_DIS
LIN {X -0.179,Y -360.651,Z 1372.695,A 0.000,B 0.000,C 90.000,E1 341.040} C_DIS
LIN {X 0.152,Y -361.861,Z 1372.684,A 0.000,B 0.000,C 90.000,E1 339.028} C_DIS
LIN {X 0.092,Y -362.508,Z 1372.671,A 0.000,B 0.000,C 90.000,E1 336.794} C_DIS
LIN {X -0.017,Y -366.061,Z 1372.642,A 0.000,B 0.000,C 90.000,E1 331.591} C_DIS
LIN {X -0.103,Y -370.617,Z 1372.607,A 0.000,B 0.000,C 90.000,E1 325.308} C_DIS
LIN {X -0.055,Y -371.814,Z 1372.601,A 0.000,B 0.000,C 90.000,E1 324.196} C_DIS
LIN {X 0.012,Y -377.461,Z 1372.567,A 0.000,B 0.000,C 90.000,E1 317.957} C_DIS
LIN {X -0.001,Y -377.940,Z 1372.564,A 0.000,B 0.000,C 90.000,E1 317.595} C_DIS
LIN {X 0.026,Y -378.526,Z 1372.560,A 0.000,B 0.000,C 90.000,E1 316.863} C_DIS
LIN {X 0.050,Y -384.546,Z 1372.528,A 0.000,B 0.000,C 90.000,E1 311.067} C_DIS
LIN {X 0.094,Y -384.945,Z 1372.526,A 0.000,B 0.000,C 90.000,E1 310.701} C_DIS
LIN {X 0.042,Y -390.718,Z 1372.494,A 0.000,B 0.000,C 90.000,E1 304.978} C_DIS
LIN {X 0.110,Y -391.215,Z 1372.492,A 0.000,B 0.000,C 90.000,E1 304.612} C_DIS
LIN {X -0.084,Y -396.929,Z 1372.459,A 0.000,B 0.000,C 90.000,E1 298.615} C_DIS
LIN {X 0.217,Y -401.297,Z 1372.428,A 0.000,B 0.000,C 90.000,E1 292.950} C_DIS
LIN {X -0.074,Y -401.645,Z 1372.426,A 0.000,B 0.000,C 90.000,E1 292.642} C_DIS
LIN {X 0.063,Y -404.723,Z 1372.395,A 0.000,B 0.000,C 90.000,E1 287.040} C_DIS
LIN {X 0.066,Y -406.142,Z 1372.364,A 0.000,B 0.000,C 90.000,E1 281.478} C_DIS
LIN {X 0.164,Y -405.687,Z 1372.333,A 0.000,B 0.000,C 90.000,E1 275.910} C_DIS
LIN {X -0.169,Y -403.572,Z 1372.306,A 0.000,B 0.000,C 90.000,E1 271.088} C_DIS
LIN {X 0.170,Y -403.225,Z 1372.302,A 0.000,B 0.000,C 90.000,E1 270.344} C_DIS
LIN {X 0.004,Y -399.085,Z 1372.273,A 0.000,B 0.000,C 90.000,E1 265.122} C_DIS
LIN {X -0.054,Y -398.834,Z 1372.271,A 0.000,B 0.000,C 90.000,E1 264.780} C_DIS
LIN {X -0.155,Y -393.325,Z 1372.244,A 0.000,B 0.000,C 90.000,E1 259.859} C_DIS
LIN {X 0.153,Y -392.736,Z 1372.240,A 0.000,B 0.000,C 90.000,E1 259.106} C_DIS
LIN {X -0.154,Y -386.292,Z 1372.214,A 0.000,B 0.000,C 90.000,E1 254.519} C_DIS
LIN {X -0.082,Y -385.191,Z 1372.208,A 0.000,B 0.000,C 90.000,E1 253.433} C_DIS
LIN {X -0.133,Y -383.328,Z 1372.202,A 0.000,B 0.000,C 90.000,E1 252.362} C_DIS
LIN {X 0.156,Y -376.975,Z 1372.178,A 0.000,B 0.000,C 90.000,E1 247.975} C_DIS
LIN {X -0.083,Y -376.142,Z 1372.174,A 0.000,B 0.000,C 90.000,E1 247.283} C_DIS
LIN {X 0.089,Y -368.307,Z 1372.147,A 0.000,B 0.000,C 90.000,E1 242.487} C_DIS
LIN {X -0.195,Y -366.448,Z 1372.139,A 0.000,B 0.000,C 90.000,E1 241.051} C_DIS
LIN {X -0.110,Y -365.888,Z 1372.137,A 0.000,B 0.000,C 90.000,E1 240.667} C_DIS
LIN {X -0.020,Y -359.079,Z 1372.114,A 0.000,B 0.000,C 90.000,E1 236.548} C_DIS
LIN {X 0.067,Y -356.228,Z 1372.102,A 0.000,B 0.000,C 90.000,E1 234.276} C_DIS
LIN {X -0.002,Y -355.689,Z 1372.099,A 0.000,B 0.000,C 90.000,E1 233.909} C_DIS
LIN {X -0.198,Y -348.687,Z 1372.074,A 0.000,B 0.000,C 90.000,E1 229.380} C_DIS
LIN {X -0.123,Y -346.100,Z 1372.061,A 0.000,B 0.000,C 90.000,E1 227.067} C_DIS
LIN {X 0.015,Y -339.731,Z 1372.036,A 0.000,B 0.000,C 90.000,E1 222.405} C_DIS
LIN {X 0.057,Y -336.732,Z 1372.018,A 0.000,B 0.000,C 90.000,E1 219.277} C_DIS
LIN {X -0.033,Y -330.793,Z 1371.988,A 0.000,B 0.000,C 90.000,E1 213.785} C_DIS
LIN {X 0.096,Y -329.240,Z 1371.974,A 0.000,B 0.000,C 90.000,E1 211.386} C_DIS
LIN {X 0.069,Y -324.628,Z 1371.941,A 0.000,B 0.000,C 90.000,E1 205.412} C_DIS
LIN {X -0.031,Y -323.796,Z 1371.928,A 0.000,B 0.000,C 90.000,E1 203.025} C_DIS
LIN {X -0.054,Y -322.904,Z 1371.921,A 0.000,B 0.000,C 90.000,E1 201.716} C_DIS
LIN {X -0.071,Y -322.940,Z 1371.921,A 0.000,B 0.000,C 90.000,E1 201.716} C_DIS
LIN {X 0.060,Y -344.741,Z 1371.913,A 0.000,B 0.000,C 90.000,E1 200.301} C_DIS
LIN {X -0.006,Y -367.650,Z 1371.906,A 0.000,B 0.000,C 90.000,E1 199.033} C_DIS
LIN {X -0.005,Y -392.496,Z 1371.899,A 0.000,B 0.000,C 90.000,E1 197.819} C_DIS
LIN {X -0.138,Y -421.061,Z 1371.892,A 0.000,B 0.000,C 90.000,E1 196.622} C_DIS
LIN {X 0.113,Y -440.809,Z 1371.888,A 0.000,B 0.000,C 90.000,E1 195.843} C_DIS
LIN {X 0.094,Y -444.084,Z 1371.887,A 0.000,B 0.000,C 90.000,E1 195.717} C_DIS
LIN {X -0.125,Y -445.348,Z 1371.887,A 0.000,B 0.000,C 90.000,E1 195.607} C_DIS
LIN {X -0.135,Y -446.741,Z 1371.885,A 0.000,B 0.000,C 90.000,E1 195.300} C_DIS
LIN {X 0.027,Y -447.592,Z 1371.883,A 0.000,B 0.000,C 90.000,E1 194.954} C_DIS
LIN {X -0.121,Y -448.145,Z 1371.881,A 0.000,B 0.000,C 90.000,E1 194.647} C_DIS
LIN {X 0.054,Y -448.507,Z 1371.880,A 0.000,B 0.000,C 90.000,E1 194.300} C_DIS
LIN {X 0.018,Y -449.253,Z 1371.872,A 0.000,B 0.000,C 90.000,E1 193.008} C_DIS
LIN {X 0.189,Y -449.821,Z 1371.863,A 0.000,B 0.000,C 90.000,E1 191.366} C_DIS
LIN {X -0.027,Y -450.089,Z 1371.858,A 0.000,B 0.000,C 90.000,E1 190.423} C_DIS
LIN {X -0.207,Y -450.357,Z 1371.851,A 0.000,B 0.000,C 90.000,E1 189.151} C_DIS
LIN {X 0.216,Y -450.447,Z 1371.838,A 0.000,B 0.000,C 90.000,E1 186.834} C_DIS
LIN {X 0.188,Y -450.479,Z 1371.829,A 0.000,B 0.000,C 90.000,E1 185.220} C_DIS
LIN {X 0.120,Y -450.192,Z 1371.820,A 0.000,B 0.000,C 90.000,E1 183.612} C_DIS
LIN {X 0.160,Y -449.669,Z 1371.815,A 0.000,B 0.000,C 90.000,E1 182.636} C_DIS
LIN {X -0.106,Y -448.573,Z 1371.808,A 0.000,B 0.000,C 90.000,E1 181.375} C_DIS
LIN {X -0.099,Y -447.465,Z 1371.802,A 0.000,B 0.000,C 90.000,E1 180.401} C_DIS
LIN {X -0.103,Y -445.891,Z 1371.797,A 0.000,B 0.000,C 90.000,E1 179.427} C_DIS
LIN {X 0.179,Y -444.741,Z 1371.793,A 0.000,B 0.000,C 90.000,E1 178.740} C_DIS
LIN {X 0.020,Y -443.318,Z 1371.790,A 0.000,B 0.000,C 90.000,E1 178.108} C_DIS
LIN {X -0.039,Y -440.456,Z 1371.784,A 0.000,B 0.000,C 90.000,E1 177.135} C_DIS
LIN {X 0.217,Y -438.293,Z 1371.781,A 0.000,B 0.000,C 90.000,E1 176.445} C_DIS
LIN {X -0.113,Y -437.112,Z 1371.779,A 0.000,B 0.000,C 90.000,E1 176.159} C_DIS
LIN {X -0.196,Y -432.722,Z 1371.773,A 0.000,B 0.000,C 90.000,E1 175.179} C_DIS
LIN {X -0.081,Y -430.301,Z 1371.770,A 0.000,B 0.000,C 90.000,E1 174.666} C_DIS
LIN {X 0.027,Y -428.449,Z 1371.769,A 0.000,B 0.000,C 90.000,E1 174.318} C_DIS
LIN {X 0.179,Y -424.431,Z 1371.765,A 0.000,B 0.000,C 90.000,E1 173.628} C_DIS
LIN {X -0.055,Y -417.827,Z 1371.759,A 0.000,B 0.000,C 90.000,E1 172.648} C_DIS
LIN {X 0.141,Y -408.547,Z 1371.752,A 0.000,B 0.000,C 90.000,E1 171.254} C_DIS
LIN {X 0.158,Y -395.184,Z 1371.740,A 0.000,B 0.000,C 90.000,E1 169.162} C_DIS
LIN {X 0.042,Y -388.897,Z 1371.734,A 0.000,B 0.000,C 90.000,E1 168.117} C_DIS
LIN {X 0.098,Y -384.486,Z 1371.729,A 0.000,B 0.000,C 90.000,E1 167.229} C_DIS
LIN {X 0.022,Y -383.122,Z 1371.727,A 0.000,B 0.000,C 90.000,E1 166.881} C_DIS
LIN {X 0.028,Y -382.000,Z 1371.725,A 0.000,B 0.000,C 90.000,E1 166.520} C_DIS
LIN {X -0.039,Y -381.715,Z 1371.724,A 0.000,B 0.000,C 90.000,E1 166.353} C_DIS
LIN {X -0.017,Y -381.674,Z 1371.723,A 0.000,B 0.000,C 90.000,E1 166.172} C_DIS
LIN {X -0.055,Y -381.682,Z 1371.723,A 0.000,B 0.000,C 90.000,E1 166.172} C_DIS
LIN {X 0.053,Y -383.067,Z 1371.721,A 0.000,B 0.000,C 90.000,E1 165.755} C_DIS
LIN {X -0.109,Y -385.478,Z 1371.719,A 0.000,B 0.000,C 90.000,E1 165.463} C_DIS
LIN {X -0.104,Y -386.702,Z 1371.718,A 0.000,B 0.000,C 90.000,E1 165.283} C_DIS
LIN {X 0.030,Y -392.531,Z 1371.714,A 0.000,B 0.000,C 90.000,E1 164.574} C_DIS
LIN {X -0.174,Y -400.362,Z 1371.710,A 0.000,B 0.000,C 90.000,E1 163.795} C_DIS
LIN {X -0.037,Y -414.320,Z 1371.703,A 0.000,B 0.000,C 90.000,E1 162.489} C_DIS
LIN {X 0.004,Y -441.305,Z 1371.691,A 0.000,B 0.000,C 90.000,E1 160.296} C_DIS
LIN {X 0.074,Y -453.784,Z 1371.685,A 0.000,B 0.000,C 90.000,E1 159.337} C_DIS
LIN {X 0.173,Y -461.513,Z 1371.682,A 0.000,B 0.000,C 90.000,E1 158.720} C_DIS
LIN {X 0.099,Y -470.669,Z 1371.678,A 0.000,B 0.000,C 90.000,E1 157.975} C_DIS
LIN {X -0.198,Y -479.527,Z 1371.673,A 0.000,B 0.000,C 90.000,E1 157.230} C_DIS
LIN {X -0.065,Y -488.227,Z 1371.669,A 0.000,B 0.000,C 90.000,E1 156.410} C_DIS
LIN {X -0.095,Y -495.235,Z 1371.665,A 0.000,B 0.000,C 90.000,E1 155.741} C_DIS
LIN {X -0.054,Y -503.376,Z 1371.661,A 0.000,B 0.000,C 90.000,E1 154.897} C_DIS
LIN {X 0.006,Y -511.025,Z 1371.656,A 0.000,B 0.000,C 90.000,E1 154.024} C_DIS
LIN {X 0.276,Y -517.269,Z 1371.652,A 0.000,B 0.000,C 90.000,E1 153.256} C_DIS
LIN {X 0.140,Y -522.954,Z 1371.648,A 0.000,B 0.000,C 90.000,E1 152.538} C_DIS
LIN {X 0.125,Y -526.168,Z 1371.645,A 0.000,B 0.000,C 90.000,E1 152.103} C_DIS
LIN {X 0.067,Y -530.802,Z 1371.641,A 0.000,B 0.000,C 90.000,E1 151.385} C_DIS
LIN {X 0.196,Y -533.964,Z 1371.638,A 0.000,B 0.000,C 90.000,E1 150.795} C_DIS
LIN {X -0.116,Y -536.685,Z 1371.635,A 0.000,B 0.000,C 90.000,E1 150.255} C_DIS
LIN {X -0.224,Y -540.123,Z 1371.630,A 0.000,B 0.000,C 90.000,E1 149.410} C_DIS
LIN {X -0.033,Y -542.186,Z 1371.627,A 0.000,B 0.000,C 90.000,E1 148.820} C_DIS
LIN {X -0.006,Y -543.963,Z 1371.624,A 0.000,B 0.000,C 90.000,E1 148.250} C_DIS
LIN {X 0.243,Y -546.199,Z 1371.619,A 0.000,B 0.000,C 90.000,E1 147.375} C_DIS
LIN {X 0.016,Y -547.474,Z 1371.616,A 0.000,B 0.000,C 90.000,E1 146.834} C_DIS
LIN {X -0.159,Y -549.061,Z 1371.611,A 0.000,B 0.000,C 90.000,E1 146.008} C_DIS
LIN {X -0.320,Y -550.449,Z 1371.606,A 0.000,B 0.000,C 90.000,E1 145.182} C_DIS
LIN {X -0.149,Y -551.641,Z 1371.602,A 0.000,B 0.000,C 90.000,E1 144.322} C_DIS
LIN {X -0.288,Y -552.561,Z 1371.597,A 0.000,B 0.000,C 90.000,E1 143.497} C_DIS
LIN {X -0.027,Y -553.505,Z 1371.591,A 0.000,B 0.000,C 90.000,E1 142.351} C_DIS
LIN {X -0.052,Y -554.652,Z 1371.582,A 0.000,B 0.000,C 90.000,E1 140.678} C_DIS
LIN {X -0.199,Y -555.506,Z 1371.574,A 0.000,B 0.000,C 90.000,E1 139.299} C_DIS
LIN {X 0.091,Y -556.279,Z 1371.566,A 0.000,B 0.000,C 90.000,E1 137.877} C_DIS
LIN {X -0.051,Y -556.895,Z 1371.558,A 0.000,B 0.000,C 90.000,E1 136.500} C_DIS
LIN {X 0.228,Y -557.436,Z 1371.551,A 0.000,B 0.000,C 90.000,E1 135.081} C_DIS
LIN {X -0.225,Y -558.077,Z 1371.541,A 0.000,B 0.000,C 90.000,E1 133.461} C_DIS
LIN {X 0.142,Y -558.702,Z 1371.532,A 0.000,B 0.000,C 90.000,E1 131.757} C_DIS
LIN {X 0.071,Y -559.321,Z 1371.524,A 0.000,B 0.000,C 90.000,E1 130.378} C_DIS
LIN {X -0.187,Y -559.701,Z 1371.521,A 0.000,B 0.000,C 90.000,E1 129.850} C_DIS
LIN {X -0.161,Y -560.664,Z 1371.518,A 0.000,B 0.000,C 90.000,E1 129.197} C_DIS
LIN {X 0.270,Y -561.760,Z 1371.516,A 0.000,B 0.000,C 90.000,E1 128.910} C_DIS
LIN {X -0.297,Y -563.668,Z 1371.516,A 0.000,B 0.000,C 90.000,E1 128.830} C_DIS
LIN {X -0.186,Y -565.285,Z 1371.515,A 0.000,B 0.000,C 90.000,E1 128.749} C_DIS
LIN {X -0.038,Y -571.754,Z 1371.514,A 0.000,B 0.000,C 90.000,E1 128.543} C_DIS
LIN {X -0.198,Y -575.490,Z 1371.514,A 0.000,B 0.000,C 90.000,E1 128.463} C_DIS
LIN {X -0.155,Y -581.434,Z 1371.512,A 0.000,B 0.000,C 90.000,E1 128.257} C_DIS
LIN {X -0.033,Y -587.348,Z 1371.511,A 0.000,B 0.000,C 90.000,E1 127.971} C_DIS
LIN {X -0.200,Y -593.378,Z 1371.509,A 0.000,B 0.000,C 90.000,E1 127.649} C_DIS
LIN {X 0.142,Y -598.952,Z 1371.507,A 0.000,B 0.000,C 90.000,E1 127.237} C_DIS
LIN {X -0.013,Y -604.513,Z 1371.505,A 0.000,B 0.000,C 90.000,E1 126.824} C_DIS
LIN {X -0.073,Y -608.528,Z 1371.503,A 0.000,B 0.000,C 90.000,E1 126.503} C_DIS
LIN {X 0.232,Y -613.685,Z 1371.500,A 0.000,B 0.000,C 90.000,E1 126.011} C_DIS
LIN {X -0.167,Y -619.954,Z 1371.497,A 0.000,B 0.000,C 90.000,E1 125.438} C_DIS
LIN {X -0.271,Y -626.031,Z 1371.493,A 0.000,B 0.000,C 90.000,E1 124.818} C_DIS
LIN {X 0.084,Y -630.695,Z 1371.490,A 0.000,B 0.000,C 90.000,E1 124.278} C_DIS
LIN {X -0.200,Y -638.919,Z 1371.485,A 0.000,B 0.000,C 90.000,E1 123.293} C_DIS
LIN {X 0.260,Y -643.591,Z 1371.481,A 0.000,B 0.000,C 90.000,E1 122.625} C_DIS
LIN {X 0.252,Y -648.702,Z 1371.477,A 0.000,B 0.000,C 90.000,E1 121.878} C_DIS
LIN {X 0.202,Y -651.824,Z 1371.474,A 0.000,B 0.000,C 90.000,E1 121.386} C_DIS
LIN {X -0.219,Y -653.975,Z 1371.472,A 0.000,B 0.000,C 90.000,E1 121.052} C_DIS
LIN {X 0.153,Y -657.028,Z 1371.469,A 0.000,B 0.000,C 90.000,E1 120.413} C_DIS
LIN {X 0.262,Y -660.186,Z 1371.465,A 0.000,B 0.000,C 90.000,E1 119.667} C_DIS
LIN {X -0.062,Y -661.917,Z 1371.462,A 0.000,B 0.000,C 90.000,E1 119.205} C_DIS
LIN {X 0.069,Y -662.685,Z 1371.461,A 0.000,B 0.000,C 90.000,E1 118.949} C_DIS
LIN {X -0.097,Y -664.506,Z 1371.457,A 0.000,B 0.000,C 90.000,E1 118.231} C_DIS
LIN {X 0.046,Y -664.905,Z 1371.455,A 0.000,B 0.000,C 90.000,E1 117.975} C_DIS
LIN {X -0.248,Y -665.318,Z 1371.453,A 0.000,B 0.000,C 90.000,E1 117.513} C_DIS
LIN {X 0.198,Y -665.489,Z 1371.449,A 0.000,B 0.000,C 90.000,E1 116.744} C_DIS
LIN {X 0.050,Y -665.188,Z 1371.445,A 0.000,B 0.000,C 90.000,E1 116.027} C_DIS
LIN {X 0.206,Y -664.508,Z 1371.441,A 0.000,B 0.000,C 90.000,E1 115.283} C_DIS
LIN {X -0.249,Y -664.218,Z 1371.439,A 0.000,B 0.000,C 90.000,E1 115.079} C_DIS
LIN {X -0.237,Y -663.246,Z 1371.437,A 0.000,B 0.000,C 90.000,E1 114.591} C_DIS
LIN {X -0.095,Y -662.610,Z 1371.435,A 0.000,B 0.000,C 90.000,E1 114.335} C_DIS
LIN {X 0.113,Y -660.708,Z 1371.433,A 0.000,B 0.000,C 90.000,E1 113.951} C_DIS
LIN {X 0.243,Y -659.295,Z 1371.432,A 0.000,B 0.000,C 90.000,E1 113.695} C_DIS
LIN {X 0.043,Y -658.284,Z 1371.431,A 0.000,B 0.000,C 90.000,E1 113.590} C_DIS
LIN {X 0.180,Y -653.499,Z 1371.429,A 0.000,B 0.000,C 90.000,E1 113.153} C_DIS
LIN {X -0.289,Y -651.912,Z 1371.428,A 0.000,B 0.000,C 90.000,E1 113.078} C_DIS
LIN {X 0.117,Y -642.392,Z 1371.426,A 0.000,B 0.000,C 90.000,E1 112.642} C_DIS
LIN {X -0.047,Y -640.280,Z 1371.426,A 0.000,B 0.000,C 90.000,E1 112.589} C_DIS
LIN {X -0.155,Y -625.473,Z 1371.423,A 0.000,B 0.000,C 90.000,E1 112.206} C_DIS
LIN {X -0.218,Y -625.352,Z 1371.423,A 0.000,B 0.000,C 90.000,E1 112.206} C_DIS
LIN {X -0.279,Y -633.871,Z 1371.418,A 0.000,B 0.000,C 90.000,E1 111.280} C_DIS
LIN {X 0.142,Y -638.228,Z 1371.415,A 0.000,B 0.000,C 90.000,E1 110.737} C_DIS
LIN {X 0.022,Y -642.936,Z 1371.412,A 0.000,B 0.000,C 90.000,E1 110.120} C_DIS
LIN {X -0.064,Y -646.966,Z 1371.408,A 0.000,B 0.000,C 90.000,E1 109.504} C_DIS
LIN {X -0.335,Y -650.413,Z 1371.405,A 0.000,B 0.000,C 90.000,E1 108.906} C_DIS
LIN {X 0.158,Y -655.251,Z 1371.399,A 0.000,B 0.000,C 90.000,E1 107.873} C_DIS
LIN {X -0.083,Y -657.545,Z 1371.397,A 0.000,B 0.000,C 90.000,E1 107.402} C_DIS
LIN {X -0.116,Y -659.689,Z 1371.394,A 0.000,B 0.000,C 90.000,E1 106.913} C_DIS
LIN {X -0.326,Y -661.571,Z 1371.391,A 0.000,B 0.000,C 90.000,E1 106.441} C_DIS
LIN {X 0.203,Y -663.980,Z 1371.387,A 0.000,B 0.000,C 90.000,E1 105.662} C_DIS
LIN {X -0.061,Y -665.754,Z 1371.383,A 0.000,B 0.000,C 90.000,E1 104.954} C_DIS
LIN {X -0.225,Y -666.711,Z 1371.380,A 0.000,B 0.000,C 90.000,E1 104.481} C_DIS
LIN {X -0.382,Y -667.429,Z 1371.378,A 0.000,B 0.000,C 90.000,E1 104.008} C_DIS
LIN {X 0.040,Y -668.115,Z 1371.374,A 0.000,B 0.000,C 90.000,E1 103.244} C_DIS
LIN {X -0.107,Y -668.304,Z 1371.371,A 0.000,B 0.000,C 90.000,E1 102.771} C_DIS
LIN {X 0.323,Y -668.225,Z 1371.367,A 0.000,B 0.000,C 90.000,E1 102.007} C_DIS
LIN {X 0.171,Y -667.970,Z 1371.364,A 0.000,B 0.000,C 90.000,E1 101.535} C_DIS
LIN {X -0.114,Y -667.461,Z 1371.362,A 0.000,B 0.000,C 90.000,E1 101.074} C_DIS
LIN {X 0.299,Y -666.292,Z 1371.357,A 0.000,B 0.000,C 90.000,E1 100.310} C_DIS
LIN {X 0.012,Y -665.281,Z 1371.355,A 0.000,B 0.000,C 90.000,E1 99.849} C_DIS
LIN {X 0.285,Y -663.316,Z 1371.351,A 0.000,B 0.000,C 90.000,E1 99.095} C_DIS
LIN {X 0.189,Y -662.627,Z 1371.349,A 0.000,B 0.000,C 90.000,E1 98.859} C_DIS
LIN {X -0.221,Y -660.014,Z 1371.345,A 0.000,B 0.000,C 90.000,E1 98.163} C_DIS
LIN {X 0.114,Y -658.069,Z 1371.343,A 0.000,B 0.000,C 90.000,E1 97.644} C_DIS
LIN {X 0.309,Y -654.678,Z 1371.339,A 0.000,B 0.000,C 90.000,E1 96.891} C_DIS
LIN {X -0.009,Y -652.817,Z 1371.336,A 0.000,B 0.000,C 90.000,E1 96.549} C_DIS
LIN {X 0.012,Y -647.916,Z 1371.332,A 0.000,B 0.000,C 90.000,E1 95.682} C_DIS
LIN {X -0.155,Y -641.719,Z 1371.326,A 0.000,B 0.000,C 90.000,E1 94.702} C_DIS
LIN {X -0.125,Y -637.540,Z 1371.323,A 0.000,B 0.000,C 90.000,E1 94.073} C_DIS
LIN {X -0.080,Y -632.735,Z 1371.319,A 0.000,B 0.000,C 90.000,E1 93.440} C_DIS
LIN {X 0.055,Y -628.284,Z 1371.316,A 0.000,B 0.000,C 90.000,E1 92.922} C_DIS
LIN {X 0.102,Y -622.091,Z 1371.313,A 0.000,B 0.000,C 90.000,E1 92.293} C_DIS
LIN {X 0.283,Y -615.737,Z 1371.309,A 0.000,B 0.000,C 90.000,E1 91.661} C_DIS
LIN {X 0.032,Y -610.455,Z 1371.307,A 0.000,B 0.000,C 90.000,E1 91.203} C_DIS
LIN {X -0.021,Y -606.009,Z 1371.305,A 0.000,B 0.000,C 90.000,E1 90.859} C_DIS
LIN {X 0.101,Y -603.184,Z 1371.304,A 0.000,B 0.000,C 90.000,E1 90.630} C_DIS
LIN {X -0.151,Y -598.217,Z 1371.302,A 0.000,B 0.000,C 90.000,E1 90.344} C_DIS
LIN {X 0.286,Y -594.993,Z 1371.301,A 0.000,B 0.000,C 90.000,E1 90.115} C_DIS
LIN {X -0.281,Y -588.030,Z 1371.299,A 0.000,B 0.000,C 90.000,E1 89.828} C_DIS
LIN {X 0.234,Y -581.150,Z 1371.297,A 0.000,B 0.000,C 90.000,E1 89.484} C_DIS
LIN {X 0.041,Y -578.322,Z 1371.297,A 0.000,B 0.000,C 90.000,E1 89.370} C_DIS
LIN {X -0.032,Y -574.182,Z 1371.295,A 0.000,B 0.000,C 90.000,E1 89.026} C_DIS
LIN {X -0.070,Y -574.166,Z 1371.295,A 0.000,B 0.000,C 90.000,E1 89.026} C_DIS
LIN {X -0.122,Y -573.693,Z 1371.294,A 0.000,B 0.000,C 90.000,E1 88.854} C_DIS
LIN {X 0.237,Y -573.562,Z 1371.293,A 0.000,B 0.000,C 90.000,E1 88.682} C_DIS
LIN {X 0.015,Y -573.860,Z 1371.289,A 0.000,B 0.000,C 90.000,E1 87.993} C_DIS
LIN {X -0.245,Y -575.205,Z 1371.280,A 0.000,B 0.000,C 90.000,E1 86.388} C_DIS
LIN {X 0.233,Y -577.953,Z 1371.265,A 0.000,B 0.000,C 90.000,E1 83.628} C_DIS
LIN {X -0.005,Y -579.571,Z 1371.257,A 0.000,B 0.000,C 90.000,E1 82.299} C_DIS
LIN {X 0.008,Y -581.520,Z 1371.248,A 0.000,B 0.000,C 90.000,E1 80.679} C_DIS
LIN {X -0.084,Y -583.095,Z 1371.241,A 0.000,B 0.000,C 90.000,E1 79.342} C_DIS
LIN {X 0.206,Y -584.713,Z 1371.232,A 0.000,B 0.000,C 90.000,E1 77.701} C_DIS
LIN {X 0.038,Y -585.672,Z 1371.226,A 0.000,B 0.000,C 90.000,E1 76.645} C_DIS
LIN {X -0.052,Y -586.892,Z 1371.217,A 0.000,B 0.000,C 90.000,E1 75.046} C_DIS
LIN {X 0.197,Y -587.773,Z 1371.209,A 0.000,B 0.000,C 90.000,E1 73.685} C_DIS
LIN {X -0.261,Y -588.802,Z 1371.201,A 0.000,B 0.000,C 90.000,E1 72.127} C_DIS
LIN {X -0.192,Y -589.492,Z 1371.193,A 0.000,B 0.000,C 90.000,E1 70.786} C_DIS
LIN {X 0.121,Y -590.448,Z 1371.184,A 0.000,B 0.000,C 90.000,E1 69.156} C_DIS
LIN {X -0.013,Y -591.595,Z 1371.174,A 0.000,B 0.000,C 90.000,E1 67.305} C_DIS
LIN {X 0.011,Y -592.612,Z 1371.167,A 0.000,B 0.000,C 90.000,E1 65.973} C_DIS
LIN {X -0.185,Y -593.755,Z 1371.159,A 0.000,B 0.000,C 90.000,E1 64.665} C_DIS
LIN {X 0.060,Y -594.944,Z 1371.150,A 0.000,B 0.000,C 90.000,E1 63.050} C_DIS
LIN {X 0.163,Y -596.655,Z 1371.139,A 0.000,B 0.000,C 90.000,E1 60.923} C_DIS
LIN {X 0.023,Y -597.878,Z 1371.131,A 0.000,B 0.000,C 90.000,E1 59.616} C_DIS
LIN {X -0.310,Y -599.123,Z 1371.124,A 0.000,B 0.000,C 90.000,E1 58.329} C_DIS
LIN {X -0.023,Y -600.180,Z 1371.118,A 0.000,B 0.000,C 90.000,E1 57.248} C_DIS
LIN {X 0.020,Y -601.377,Z 1371.111,A 0.000,B 0.000,C 90.000,E1 55.928} C_DIS
LIN {X -0.011,Y -602.826,Z 1371.102,A 0.000,B 0.000,C 90.000,E1 54.356} C_DIS
LIN {X -0.391,Y -604.506,Z 1371.092,A 0.000,B 0.000,C 90.000,E1 52.557} C_DIS
LIN {X 0.178,Y -605.312,Z 1371.086,A 0.000,B 0.000,C 90.000,E1 51.457} C_DIS
LIN {X 0.170,Y -606.054,Z 1371.079,A 0.000,B 0.000,C 90.000,E1 50.150} C_DIS
LIN {X 0.094,Y -606.698,Z 1371.072,A 0.000,B 0.000,C 90.000,E1 48.852} C_DIS
LIN {X 0.225,Y -607.052,Z 1371.066,A 0.000,B 0.000,C 90.000,E1 47.796} C_DIS
LIN {X -0.284,Y -607.304,Z 1371.058,A 0.000,B 0.000,C 90.000,E1 46.539} C_DIS
LIN {X 0.066,Y -607.342,Z 1371.051,A 0.000,B 0.000,C 90.000,E1 45.202} C_DIS
LIN {X -0.256,Y -607.161,Z 1371.045,A 0.000,B 0.000,C 90.000,E1 44.190} C_DIS
LIN {X -0.155,Y -606.797,Z 1371.040,A 0.000,B 0.000,C 90.000,E1 43.137} C_DIS
LIN {X 0.036,Y -606.018,Z 1371.031,A 0.000,B 0.000,C 90.000,E1 41.553} C_DIS
LIN {X -0.296,Y -605.438,Z 1371.025,A 0.000,B 0.000,C 90.000,E1 40.539} C_DIS
LIN {X -0.184,Y -604.754,Z 1371.019,A 0.000,B 0.000,C 90.000,E1 39.483} C_DIS
LIN {X -0.206,Y -603.691,Z 1371.012,A 0.000,B 0.000,C 90.000,E1 38.177} C_DIS
LIN {X -0.243,Y -602.403,Z 1371.005,A 0.000,B 0.000,C 90.000,E1 36.870} C_DIS
LIN {X -0.324,Y -601.406,Z 1371.000,A 0.000,B 0.000,C 90.000,E1 36.091} C_DIS
LIN {X -0.171,Y -599.701,Z 1370.995,A 0.000,B 0.000,C 90.000,E1 35.025} C_DIS
LIN {X -0.029,Y -598.642,Z 1370.992,A 0.000,B 0.000,C 90.000,E1 34.485} C_DIS
LIN {X 0.076,Y -596.376,Z 1370.986,A 0.000,B 0.000,C 90.000,E1 33.420} C_DIS
LIN {X 0.096,Y -594.463,Z 1370.981,A 0.000,B 0.000,C 90.000,E1 32.625} C_DIS
LIN {X 0.208,Y -593.038,Z 1370.978,A 0.000,B 0.000,C 90.000,E1 32.084} C_DIS
LIN {X -0.103,Y -589.863,Z 1370.973,A 0.000,B 0.000,C 90.000,E1 31.052} C_DIS
LIN {X -0.259,Y -585.990,Z 1370.967,A 0.000,B 0.000,C 90.000,E1 30.001} C_DIS
LIN {X 0.173,Y -582.732,Z 1370.962,A 0.000,B 0.000,C 90.000,E1 29.155} C_DIS
LIN {X 0.061,Y -579.036,Z 1370.958,A 0.000,B 0.000,C 90.000,E1 28.359} C_DIS
LIN {X -0.295,Y -575.673,Z 1370.954,A 0.000,B 0.000,C 90.000,E1 27.719} C_DIS
LIN {X -0.064,Y -570.546,Z 1370.949,A 0.000,B 0.000,C 90.000,E1 26.744} C_DIS
LIN {X -0.065,Y -565.753,Z 1370.944,A 0.000,B 0.000,C 90.000,E1 25.924} C_DIS
LIN {X 0.222,Y -561.397,Z 1370.940,A 0.000,B 0.000,C 90.000,E1 25.207} C_DIS
LIN {X -0.177,Y -557.679,Z 1370.937,A 0.000,B 0.000,C 90.000,E1 24.695} C_DIS
LIN {X 0.188,Y -551.691,Z 1370.932,A 0.000,B 0.000,C 90.000,E1 23.823} C_DIS
LIN {X 0.106,Y -546.310,Z 1370.929,A 0.000,B 0.000,C 90.000,E1 23.131} C_DIS
LIN {X -0.235,Y -540.492,Z 1370.925,A 0.000,B 0.000,C 90.000,E1 22.461} C_DIS
LIN {X 0.009,Y -533.206,Z 1370.920,A 0.000,B 0.000,C 90.000,E1 21.589} C_DIS
LIN {X -0.035,Y -522.933,Z 1370.914,A 0.000,B 0.000,C 90.000,E1 20.482} C_DIS
LIN {X -0.138,Y -512.404,Z 1370.908,A 0.000,B 0.000,C 90.000,E1 19.396} C_DIS
LIN {X 0.047,Y -503.200,Z 1370.902,A 0.000,B 0.000,C 90.000,E1 18.417} C_DIS
LIN {X 0.231,Y -492.144,Z 1370.896,A 0.000,B 0.000,C 90.000,E1 17.275} C_DIS
LIN {X 0.181,Y -478.149,Z 1370.889,A 0.000,B 0.000,C 90.000,E1 15.898} C_DIS
LIN {X 0.070,Y -466.890,Z 1370.882,A 0.000,B 0.000,C 90.000,E1 14.773} C_DIS
LIN {X 0.047,Y -456.938,Z 1370.877,A 0.000,B 0.000,C 90.000,E1 13.772} C_DIS
LIN {X 0.114,Y -439.984,Z 1370.867,A 0.000,B 0.000,C 90.000,E1 12.007} C_DIS
LIN {X -0.123,Y -430.437,Z 1370.861,A 0.000,B 0.000,C 90.000,E1 11.007} C_DIS
LIN {X -0.160,Y -415.156,Z 1370.851,A 0.000,B 0.000,C 90.000,E1 9.265} C_DIS
LIN {X 0.147,Y -402.640,Z 1370.843,A 0.000,B 0.000,C 90.000,E1 7.757} C_DIS
LIN {X -0.031,Y -396.969,Z 1370.840,A 0.000,B 0.000,C 90.000,E1 7.125} C_DIS
LIN {X -0.011,Y -392.915,Z 1370.836,A 0.000,B 0.000,C 90.000,E1 6.549} C_DIS
LIN {X 0.105,Y -392.183,Z 1370.836,A 0.000,B 0.000,C 90.000,E1 6.372} C_DIS
LIN {X 0.067,Y -392.183,Z 1370.835,A 0.000,B 0.000,C 90.000,E1 6.372} C_DIS
LIN {X 0.123,Y -394.079,Z 1370.834,A 0.000,B 0.000,C 90.000,E1 6.087} C_DIS
LIN {X 0.135,Y -398.611,Z 1370.832,A 0.000,B 0.000,C 90.000,E1 5.682} C_DIS
LIN {X -0.051,Y -404.632,Z 1370.829,A 0.000,B 0.000,C 90.000,E1 5.277} C_DIS
LIN {X 0.078,Y -410.912,Z 1370.827,A 0.000,B 0.000,C 90.000,E1 4.759} C_DIS
LIN {X -0.054,Y -417.071,Z 1370.824,A 0.000,B 0.000,C 90.000,E1 4.245} C_DIS
LIN {X 0.027,Y -424.174,Z 1370.819,A 0.000,B 0.000,C 90.000,E1 3.498} C_DIS
LIN {X 0.118,Y -430.855,Z 1370.815,A 0.000,B 0.000,C 90.000,E1 2.694} C_DIS
LIN {X 0.003,Y -438.457,Z 1370.810,A 0.000,B 0.000,C 90.000,E1 1.718} C_DIS
LIN {X -0.161,Y -444.559,Z 1370.805,A 0.000,B 0.000,C 90.000,E1 0.917} C_DIS
LIN {X 0.000,Y -450.826,Z 1370.800,A 0.000,B 0.000,C 90.000,E1 360.000} C_DIS
LIN {X 0.054,Y -456.375,Z 1370.795,A 0.000,B 0.000,C 90.000,E1 359.141} C_DIS
LIN {X -0.035,Y -460.363,Z 1370.792,A 0.000,B 0.000,C 90.000,E1 358.511} C_DIS
LIN {X 0.029,Y -464.936,Z 1370.787,A 0.000,B 0.000,C 90.000,E1 357.707} C_DIS
LIN {X 0.116,Y -469.230,Z 1370.783,A 0.000,B 0.000,C 90.000,E1 356.906} C_DIS
LIN {X -0.202,Y -473.168,Z 1370.779,A 0.000,B 0.000,C 90.000,E1 356.159} C_DIS
LIN {X -0.012,Y -476.791,Z 1370.774,A 0.000,B 0.000,C 90.000,E1 355.355} C_DIS
LIN {X -0.081,Y -480.719,Z 1370.769,A 0.000,B 0.000,C 90.000,E1 354.432} C_DIS
LIN {X 0.044,Y -483.143,Z 1370.766,A 0.000,B 0.000,C 90.000,E1 353.799} C_DIS
LIN {X 0.045,Y -486.515,Z 1370.760,A 0.000,B 0.000,C 90.000,E1 352.875} C_DIS
LIN {X 0.084,Y -489.522,Z 1370.755,A 0.000,B 0.000,C 90.000,E1 351.951} C_DIS
LIN {X 0.155,Y -492.150,Z 1370.750,A 0.000,B 0.000,C 90.000,E1 351.027} C_DIS
LIN {X -0.154,Y -494.469,Z 1370.745,A 0.000,B 0.000,C 90.000,E1 350.151} C_DIS
LIN {X 0.053,Y -496.633,Z 1370.740,A 0.000,B 0.000,C 90.000,E1 349.218} C_DIS
LIN {X -0.202,Y -498.525,Z 1370.735,A 0.000,B 0.000,C 90.000,E1 348.342} C_DIS
LIN {X 0.049,Y -500.173,Z 1370.730,A 0.000,B 0.000,C 90.000,E1 347.409} C_DIS
LIN {X -0.102,Y -500.968,Z 1370.727,A 0.000,B 0.000,C 90.000,E1 346.825} C_DIS
LIN {X -0.059,Y -501.144,Z 1370.725,A 0.000,B 0.000,C 90.000,E1 346.520} C_DIS
LIN {X -0.130,Y -501.092,Z 1370.724,A 0.000,B 0.000,C 90.000,E1 346.228} C_DIS
LIN {X -0.202,Y -500.647,Z 1370.722,A 0.000,B 0.000,C 90.000,E1 345.936} C_DIS
LIN {X 0.066,Y -500.162,Z 1370.721,A 0.000,B 0.000,C 90.000,E1 345.755} C_DIS
LIN {X -0.274,Y -499.274,Z 1370.720,A 0.000,B 0.000,C 90.000,E1 345.644} C_DIS
LIN {X 0.181,Y -496.675,Z 1370.719,A 0.000,B 0.000,C 90.000,E1 345.463} C_DIS
LIN {X 0.180,Y -462.803,Z 1370.714,A 0.000,B 0.000,C 90.000,E1 344.393} C_DIS
LIN {X 0.025,Y -431.400,Z 1370.707,A 0.000,B 0.000,C 90.000,E1 343.268} C_DIS
LIN {X -0.122,Y -403.682,Z 1370.701,A 0.000,B 0.000,C 90.000,E1 342.127} C_DIS
LIN {X -0.058,Y -379.610,Z 1370.694,A 0.000,B 0.000,C 90.000,E1 340.967} C_DIS
LIN {X -0.215,Y -361.247,Z 1370.689,A 0.000,B 0.000,C 90.000,E1 340.007} C_DIS
LIN {X 0.104,Y -361.240,Z 1370.689,A 0.000,B 0.000,C 90.000,E1 339.953} C_DIS
LIN {X 0.134,Y -361.825,Z 1370.684,A 0.000,B 0.000,C 90.000,E1 339.082} C_DIS
LIN {X 0.112,Y -362.059,Z 1370.680,A 0.000,B 0.000,C 90.000,E1 338.337} C_DIS
LIN {X -0.017,Y -366.011,Z 1370.642,A 0.000,B 0.000,C 90.000,E1 331.641} C_DIS
LIN {X -0.177,Y -366.401,Z 1370.638,A 0.000,B 0.000,C 90.000,E1 330.923} C_DIS
LIN {X -0.022,Y -371.393,Z 1370.603,A 0.000,B 0.000,C 90.000,E1 324.609} C_DIS
LIN {X -0.033,Y -371.786,Z 1370.601,A 0.000,B 0.000,C 90.000,E1 324.242} C_DIS
LIN {X 0.057,Y -377.398,Z 1370.567,A 0.000,B 0.000,C 90.000,E1 318.000} C_DIS
LIN {X -0.196,Y -378.254,Z 1370.563,A 0.000,B 0.000,C 90.000,E1 317.310} C_DIS
LIN {X 0.080,Y -383.982,Z 1370.531,A 0.000,B 0.000,C 90.000,E1 311.472} C_DIS
LIN {X -0.121,Y -384.914,Z 1370.526,A 0.000,B 0.000,C 90.000,E1 310.782} C_DIS
LIN {X 0.051,Y -390.652,Z 1370.495,A 0.000,B 0.000,C 90.000,E1 305.025} C_DIS
LIN {X -0.106,Y -391.148,Z 1370.493,A 0.000,B 0.000,C 90.000,E1 304.692} C_DIS
LIN {X 0.061,Y -392.156,Z 1370.485,A 0.000,B 0.000,C 90.000,E1 303.245} C_DIS
LIN {X 0.247,Y -396.866,Z 1370.459,A 0.000,B 0.000,C 90.000,E1 298.615} C_DIS
LIN {X -0.200,Y -397.299,Z 1370.455,A 0.000,B 0.000,C 90.000,E1 297.975} C_DIS
LIN {X -0.112,Y -401.620,Z 1370.426,A 0.000,B 0.000,C 90.000,E1 292.695} C_DIS
LIN {X 0.009,Y -404.686,Z 1370.395,A 0.000,B 0.000,C 90.000,E1 287.094} C_DIS
LIN {X -0.190,Y -404.734,Z 1370.389,A 0.000,B 0.000,C 90.000,E1 286.079} C_DIS
LIN {X 0.001,Y -406.117,Z 1370.364,A 0.000,B 0.000,C 90.000,E1 281.535} C_DIS
LIN {X 0.021,Y -405.949,Z 1370.360,A 0.000,B 0.000,C 90.000,E1 280.838} C_DIS
LIN {X 0.094,Y -405.687,Z 1370.333,A 0.000,B 0.000,C 90.000,E1 275.967} C_DIS
LIN {X 0.131,Y -403.478,Z 1370.304,A 0.000,B 0.000,C 90.000,E1 270.745} C_DIS
LIN {X 0.098,Y -403.268,Z 1370.302,A 0.000,B 0.000,C 90.000,E1 270.401} C_DIS
LIN {X -0.120,Y -398.897,Z 1370.271,A 0.000,B 0.000,C 90.000,E1 264.837} C_DIS
LIN {X 0.174,Y -393.362,Z 1370.244,A 0.000,B 0.000,C 90.000,E1 259.859} C_DIS
LIN {X 0.096,Y -392.800,Z 1370.240,A 0.000,B 0.000,C 90.000,E1 259.162} C_DIS
LIN {X -0.199,Y -386.345,Z 1370.214,A 0.000,B 0.000,C 90.000,E1 254.574} C_DIS
LIN {X 0.135,Y -385.238,Z 1370.208,A 0.000,B 0.000,C 90.000,E1 253.449} C_DIS
LIN {X 0.156,Y -384.710,Z 1370.206,A 0.000,B 0.000,C 90.000,E1 253.087} C_DIS
LIN {X 0.014,Y -377.932,Z 1370.182,A 0.000,B 0.000,C 90.000,E1 248.773} C_DIS
LIN {X 0.096,Y -376.199,Z 1370.174,A 0.000,B 0.000,C 90.000,E1 247.305} C_DIS
LIN {X -0.060,Y -373.549,Z 1370.166,A 0.000,B 0.000,C 90.000,E1 245.869} C_DIS
LIN {X 0.038,Y -366.948,Z 1370.141,A 0.000,B 0.000,C 90.000,E1 241.435} C_DIS
LIN {X -0.109,Y -365.984,Z 1370.137,A 0.000,B 0.000,C 90.000,E1 240.717} C_DIS
LIN {X 0.100,Y -359.151,Z 1370.115,A 0.000,B 0.000,C 90.000,E1 236.580} C_DIS
LIN {X 0.095,Y -356.285,Z 1370.102,A 0.000,B 0.000,C 90.000,E1 234.322} C_DIS
LIN {X -0.182,Y -355.781,Z 1370.100,A 0.000,B 0.000,C 90.000,E1 233.989} C_DIS
LIN {X 0.117,Y -348.751,Z 1370.074,A 0.000,B 0.000,C 90.000,E1 229.380} C_DIS
LIN {X -0.044,Y -346.152,Z 1370.062,A 0.000,B 0.000,C 90.000,E1 227.106} C_DIS
LIN {X 0.199,Y -345.012,Z 1370.057,A 0.000,B 0.000,C 90.000,E1 226.296} C_DIS
LIN {X -0.105,Y -338.552,Z 1370.029,A 0.000,B 0.000,C 90.000,E1 221.310} C_DIS
LIN {X -0.106,Y -336.801,Z 1370.019,A 0.000,B 0.000,C 90.000,E1 219.358} C_DIS
LIN {X 0.001,Y -330.835,Z 1369.988,A 0.000,B 0.000,C 90.000,E1 213.833} C_DIS
LIN {X -0.048,Y -329.278,Z 1369.975,A 0.000,B 0.000,C 90.000,E1 211.465} C_DIS
LIN {X 0.083,Y -324.653,Z 1369.942,A 0.000,B 0.000,C 90.000,E1 205.463} C_DIS
LIN {X -0.022,Y -323.825,Z 1369.928,A 0.000,B 0.000,C 90.000,E1 203.078} C_DIS
LIN {X -0.188,Y -323.683,Z 1369.927,A 0.000,B 0.000,C 90.000,E1 202.898} C_DIS
LIN {X -0.206,Y -323.725,Z 1369.927,A 0.000,B 0.000,C 90.000,E1 202.898} C_DIS
LIN {X -0.178,Y -343.707,Z 1369.920,A 0.000,B 0.000,C 90.000,E1 201.535} C_DIS
LIN {X 0.194,Y -366.446,Z 1369.912,A 0.000,B 0.000,C 90.000,E1 200.120} C_DIS
LIN {X 0.082,Y -391.131,Z 1369.905,A 0.000,B 0.000,C 90.000,E1 198.852} C_DIS
LIN {X 0.098,Y -417.763,Z 1369.898,A 0.000,B 0.000,C 90.000,E1 197.638} C_DIS
LIN {X -0.217,Y -442.747,Z 1369.893,A 0.000,B 0.000,C 90.000,E1 196.677} C_DIS
LIN {X 0.146,Y -445.417,Z 1369.892,A 0.000,B 0.000,C 90.000,E1 196.496} C_DIS
LIN {X 0.211,Y -446.635,Z 1369.891,A 0.000,B 0.000,C 90.000,E1 196.315} C_DIS
LIN {X -0.201,Y -447.356,Z 1369.890,A 0.000,B 0.000,C 90.000,E1 196.205} C_DIS
LIN {X -0.059,Y -447.899,Z 1369.889,A 0.000,B 0.000,C 90.000,E1 196.024} C_DIS
LIN {X 0.231,Y -448.686,Z 1369.887,A 0.000,B 0.000,C 90.000,E1 195.662} C_DIS
LIN {X -0.029,Y -449.211,Z 1369.885,A 0.000,B 0.000,C 90.000,E1 195.371} C_DIS
LIN {X 0.011,Y -449.760,Z 1369.882,A 0.000,B 0.000,C 90.000,E1 194.717} C_DIS
LIN {X -0.145,Y -450.780,Z 1369.873,A 0.000,B 0.000,C 90.000,E1 193.119} C_DIS
LIN {X 0.049,Y -451.415,Z 1369.864,A 0.000,B 0.000,C 90.000,E1 191.478} C_DIS
LIN {X 0.173,Y -451.998,Z 1369.855,A 0.000,B 0.000,C 90.000,E1 189.849} C_DIS
LIN {X -0.144,Y -452.188,Z 1369.846,A 0.000,B 0.000,C 90.000,E1 188.276} C_DIS
LIN {X -0.140,Y -452.383,Z 1369.837,A 0.000,B 0.000,C 90.000,E1 186.663} C_DIS
LIN {X 0.167,Y -452.515,Z 1369.830,A 0.000,B 0.000,C 90.000,E1 185.334} C_DIS
LIN {X 0.136,Y -452.243,Z 1369.821,A 0.000,B 0.000,C 90.000,E1 183.726} C_DIS
LIN {X 0.199,Y -451.886,Z 1369.815,A 0.000,B 0.000,C 90.000,E1 182.751} C_DIS
LIN {X 0.129,Y -450.732,Z 1369.807,A 0.000,B 0.000,C 90.000,E1 181.146} C_DIS
LIN {X 0.001,Y -450.081,Z 1369.803,A 0.000,B 0.000,C 90.000,E1 180.516} C_DIS
LIN {X 0.027,Y -448.655,Z 1369.797,A 0.000,B 0.000,C 90.000,E1 179.542} C_DIS
LIN {X -0.114,Y -447.508,Z 1369.794,A 0.000,B 0.000,C 90.000,E1 178.912} C_DIS
LIN {X -0.108,Y -445.439,Z 1369.788,A 0.000,B 0.000,C 90.000,E1 177.936} C_DIS
LIN {X 0.169,Y -443.713,Z 1369.785,A 0.000,B 0.000,C 90.000,E1 177.249} C_DIS
LIN {X 0.132,Y -440.516,Z 1369.779,A 0.000,B 0.000,C 90.000,E1 176.274} C_DIS
LIN {X 0.000,Y -437.202,Z 1369.775,A 0.000,B 0.000,C 90.000,E1 175.469} C_DIS
LIN {X -0.083,Y -432.605,Z 1369.769,A 0.000,B 0.000,C 90.000,E1 174.489} C_DIS
LIN {X 0.161,Y -426.704,Z 1369.764,A 0.000,B 0.000,C 90.000,E1 173.457} C_DIS
LIN {X 0.006,Y -420.187,Z 1369.758,A 0.000,B 0.000,C 90.000,E1 172.470} C_DIS
LIN {X 0.193,Y -412.068,Z 1369.752,A 0.000,B 0.000,C 90.000,E1 171.254} C_DIS
LIN {X -0.145,Y -397.526,Z 1369.739,A 0.000,B 0.000,C 90.000,E1 169.050} C_DIS
LIN {X -0.197,Y -389.189,Z 1369.731,A 0.000,B 0.000,C 90.000,E1 167.645} C_DIS
LIN {X 0.157,Y -385.073,Z 1369.726,A 0.000,B 0.000,C 90.000,E1 166.700} C_DIS
LIN {X 0.062,Y -383.507,Z 1369.723,A 0.000,B 0.000,C 90.000,E1 166.061} C_DIS
LIN {X 0.026,Y -383.508,Z 1369.723,A 0.000,B 0.000,C 90.000,E1 166.061} C_DIS
LIN {X 0.036,Y -384.229,Z 1369.721,A 0.000,B 0.000,C 90.000,E1 165.700} C_DIS
LIN {X -0.001,Y -384.244,Z 1369.721,A 0.000,B 0.000,C 90.000,E1 165.700} C_DIS
LIN {X -0.156,Y -387.900,Z 1369.718,A 0.000,B 0.000,C 90.000,E1 165.172} C_DIS
LIN {X -0.087,Y -392.203,Z 1369.715,A 0.000,B 0.000,C 90.000,E1 164.629} C_DIS
LIN {X 0.153,Y -399.012,Z 1369.711,A 0.000,B 0.000,C 90.000,E1 163.866} C_DIS
LIN {X 0.011,Y -412.818,Z 1369.703,A 0.000,B 0.000,C 90.000,E1 162.598} C_DIS
LIN {X -0.073,Y -431.662,Z 1369.695,A 0.000,B 0.000,C 90.000,E1 161.040} C_DIS
LIN {X -0.067,Y -450.786,Z 1369.687,A 0.000,B 0.000,C 90.000,E1 159.571} C_DIS
LIN {X 0.078,Y -459.902,Z 1369.683,A 0.000,B 0.000,C 90.000,E1 158.847} C_DIS
LIN {X 0.045,Y -467.536,Z 1369.679,A 0.000,B 0.000,C 90.000,E1 158.230} C_DIS
LIN {X 0.205,Y -471.884,Z 1369.677,A 0.000,B 0.000,C 90.000,E1 157.847} C_DIS
LIN {X -0.129,Y -480.802,Z 1369.673,A 0.000,B 0.000,C 90.000,E1 157.102} C_DIS
LIN {X -0.128,Y -490.658,Z 1369.668,A 0.000,B 0.000,C 90.000,E1 156.177} C_DIS
LIN {X 0.038,Y -496.280,Z 1369.665,A 0.000,B 0.000,C 90.000,E1 155.613} C_DIS
LIN {X -0.058,Y -503.103,Z 1369.661,A 0.000,B 0.000,C 90.000,E1 154.921} C_DIS
LIN {X 0.210,Y -510.812,Z 1369.656,A 0.000,B 0.000,C 90.000,E1 154.024} C_DIS
LIN {X 0.024,Y -515.787,Z 1369.653,A 0.000,B 0.000,C 90.000,E1 153.461} C_DIS
LIN {X 0.206,Y -519.370,Z 1369.650,A 0.000,B 0.000,C 90.000,E1 152.999} C_DIS
LIN {X -0.070,Y -525.911,Z 1369.645,A 0.000,B 0.000,C 90.000,E1 152.153} C_DIS
LIN {X -0.129,Y -530.604,Z 1369.641,A 0.000,B 0.000,C 90.000,E1 151.435} C_DIS
LIN {X 0.000,Y -533.749,Z 1369.638,A 0.000,B 0.000,C 90.000,E1 150.845} C_DIS
LIN {X 0.013,Y -537.074,Z 1369.634,A 0.000,B 0.000,C 90.000,E1 150.127} C_DIS
LIN {X 0.048,Y -539.920,Z 1369.630,A 0.000,B 0.000,C 90.000,E1 149.410} C_DIS
LIN {X -0.226,Y -542.001,Z 1369.627,A 0.000,B 0.000,C 90.000,E1 148.869} C_DIS
LIN {X -0.022,Y -543.748,Z 1369.624,A 0.000,B 0.000,C 90.000,E1 148.280} C_DIS
LIN {X -0.242,Y -546.016,Z 1369.619,A 0.000,B 0.000,C 90.000,E1 147.454} C_DIS
LIN {X 0.022,Y -547.845,Z 1369.614,A 0.000,B 0.000,C 90.000,E1 146.580} C_DIS
LIN {X -0.105,Y -549.827,Z 1369.608,A 0.000,B 0.000,C 90.000,E1 145.468} C_DIS
LIN {X 0.056,Y -551.075,Z 1369.604,A 0.000,B 0.000,C 90.000,E1 144.609} C_DIS
LIN {X -0.087,Y -552.073,Z 1369.599,A 0.000,B 0.000,C 90.000,E1 143.783} C_DIS
LIN {X 0.167,Y -553.108,Z 1369.593,A 0.000,B 0.000,C 90.000,E1 142.637} C_DIS
LIN {X 0.068,Y -554.101,Z 1369.585,A 0.000,B 0.000,C 90.000,E1 141.251} C_DIS
LIN {X -0.020,Y -554.984,Z 1369.577,A 0.000,B 0.000,C 90.000,E1 139.865} C_DIS
LIN {X 0.276,Y -555.958,Z 1369.568,A 0.000,B 0.000,C 90.000,E1 138.162} C_DIS
LIN {X 0.157,Y -556.640,Z 1369.560,A 0.000,B 0.000,C 90.000,E1 136.782} C_DIS
LIN {X 0.081,Y -557.291,Z 1369.551,A 0.000,B 0.000,C 90.000,E1 135.121} C_DIS
LIN {X 0.085,Y -558.030,Z 1369.540,A 0.000,B 0.000,C 90.000,E1 133.176} C_DIS
LIN {X 0.382,Y -558.620,Z 1369.532,A 0.000,B 0.000,C 90.000,E1 131.757} C_DIS
LIN {X -0.052,Y -559.347,Z 1369.525,A 0.000,B 0.000,C 90.000,E1 130.415} C_DIS
LIN {X -0.033,Y -559.613,Z 1369.523,A 0.000,B 0.000,C 90.000,E1 130.135} C_DIS
LIN {X 0.052,Y -560.337,Z 1369.521,A 0.000,B 0.000,C 90.000,E1 129.850} C_DIS
LIN {X 0.100,Y -560.800,Z 1369.520,A 0.000,B 0.000,C 90.000,E1 129.564} C_DIS
LIN {X 0.058,Y -560.815,Z 1369.520,A 0.000,B 0.000,C 90.000,E1 129.564} C_DIS
LIN {X 0.137,Y -561.681,Z 1369.519,A 0.000,B 0.000,C 90.000,E1 129.439} C_DIS
LIN {X -0.074,Y -562.541,Z 1369.518,A 0.000,B 0.000,C 90.000,E1 129.322} C_DIS
LIN {X -0.204,Y -564.846,Z 1369.518,A 0.000,B 0.000,C 90.000,E1 129.197} C_DIS
LIN {X -0.168,Y -579.642,Z 1369.515,A 0.000,B 0.000,C 90.000,E1 128.749} C_DIS
LIN {X -0.009,Y -582.404,Z 1369.515,A 0.000,B 0.000,C 90.000,E1 128.624} C_DIS
LIN {X 0.253,Y -585.326,Z 1369.514,A 0.000,B 0.000,C 90.000,E1 128.463} C_DIS
LIN {X -0.130,Y -591.322,Z 1369.512,A 0.000,B 0.000,C 90.000,E1 128.177} C_DIS
LIN {X -0.223,Y -597.037,Z 1369.510,A 0.000,B 0.000,C 90.000,E1 127.810} C_DIS
LIN {X 0.334,Y -601.375,Z 1369.508,A 0.000,B 0.000,C 90.000,E1 127.443} C_DIS
LIN {X 0.075,Y -609.590,Z 1369.505,A 0.000,B 0.000,C 90.000,E1 126.790} C_DIS
LIN {X -0.184,Y -612.160,Z 1369.503,A 0.000,B 0.000,C 90.000,E1 126.583} C_DIS
LIN {X 0.329,Y -619.724,Z 1369.499,A 0.000,B 0.000,C 90.000,E1 125.804} C_DIS
LIN {X -0.248,Y -625.747,Z 1369.496,A 0.000,B 0.000,C 90.000,E1 125.231} C_DIS
LIN {X 0.088,Y -629.246,Z 1369.494,A 0.000,B 0.000,C 90.000,E1 124.818} C_DIS
LIN {X -0.075,Y -633.612,Z 1369.491,A 0.000,B 0.000,C 90.000,E1 124.326} C_DIS
LIN {X -0.171,Y -640.706,Z 1369.486,A 0.000,B 0.000,C 90.000,E1 123.452} C_DIS
LIN {X -0.238,Y -645.292,Z 1369.482,A 0.000,B 0.000,C 90.000,E1 122.832} C_DIS
LIN {X 0.152,Y -651.152,Z 1369.478,A 0.000,B 0.000,C 90.000,E1 121.926} C_DIS
LIN {X -0.129,Y -655.426,Z 1369.473,A 0.000,B 0.000,C 90.000,E1 121.209} C_DIS
LIN {X -0.141,Y -657.959,Z 1369.471,A 0.000,B 0.000,C 90.000,E1 120.718} C_DIS
LIN {X -0.359,Y -661.174,Z 1369.467,A 0.000,B 0.000,C 90.000,E1 120.001} C_DIS
LIN {X 0.361,Y -663.806,Z 1369.463,A 0.000,B 0.000,C 90.000,E1 119.205} C_DIS
LIN {X 0.204,Y -665.654,Z 1369.458,A 0.000,B 0.000,C 90.000,E1 118.487} C_DIS
LIN {X -0.087,Y -666.481,Z 1369.456,A 0.000,B 0.000,C 90.000,E1 118.025} C_DIS
LIN {X 0.064,Y -666.766,Z 1369.454,A 0.000,B 0.000,C 90.000,E1 117.769} C_DIS
LIN {X 0.370,Y -667.012,Z 1369.452,A 0.000,B 0.000,C 90.000,E1 117.257} C_DIS
LIN {X -0.059,Y -666.997,Z 1369.448,A 0.000,B 0.000,C 90.000,E1 116.565} C_DIS
LIN {X -0.346,Y -666.757,Z 1369.445,A 0.000,B 0.000,C 90.000,E1 116.104} C_DIS
LIN {X 0.115,Y -666.095,Z 1369.441,A 0.000,B 0.000,C 90.000,E1 115.335} C_DIS
LIN {X 0.136,Y -665.460,Z 1369.438,A 0.000,B 0.000,C 90.000,E1 114.847} C_DIS
LIN {X -0.170,Y -664.276,Z 1369.435,A 0.000,B 0.000,C 90.000,E1 114.387} C_DIS
LIN {X -0.026,Y -663.315,Z 1369.434,A 0.000,B 0.000,C 90.000,E1 114.131} C_DIS
LIN {X -0.016,Y -660.474,Z 1369.431,A 0.000,B 0.000,C 90.000,E1 113.643} C_DIS
LIN {X 0.049,Y -659.363,Z 1369.431,A 0.000,B 0.000,C 90.000,E1 113.515} C_DIS
LIN {X -0.316,Y -655.284,Z 1369.429,A 0.000,B 0.000,C 90.000,E1 113.206} C_DIS
LIN {X -0.255,Y -653.026,Z 1369.428,A 0.000,B 0.000,C 90.000,E1 113.025} C_DIS
LIN {X -0.020,Y -650.614,Z 1369.427,A 0.000,B 0.000,C 90.000,E1 112.898} C_DIS
LIN {X 0.015,Y -642.911,Z 1369.426,A 0.000,B 0.000,C 90.000,E1 112.589} C_DIS
LIN {X -0.043,Y -633.014,Z 1369.424,A 0.000,B 0.000,C 90.000,E1 112.333} C_DIS
LIN {X 0.152,Y -626.788,Z 1369.423,A 0.000,B 0.000,C 90.000,E1 112.153} C_DIS
LIN {X 0.092,Y -626.650,Z 1369.423,A 0.000,B 0.000,C 90.000,E1 112.153} C_DIS
LIN {X -0.217,Y -634.741,Z 1369.418,A 0.000,B 0.000,C 90.000,E1 111.280} C_DIS
LIN {X 0.209,Y -639.032,Z 1369.415,A 0.000,B 0.000,C 90.000,E1 110.737} C_DIS
LIN {X -0.132,Y -642.665,Z 1369.413,A 0.000,B 0.000,C 90.000,E1 110.301} C_DIS
LIN {X 0.200,Y -647.579,Z 1369.409,A 0.000,B 0.000,C 90.000,E1 109.523} C_DIS
LIN {X 0.153,Y -651.029,Z 1369.405,A 0.000,B 0.000,C 90.000,E1 108.906} C_DIS
LIN {X -0.168,Y -655.806,Z 1369.400,A 0.000,B 0.000,C 90.000,E1 107.946} C_DIS
LIN {X -0.322,Y -659.142,Z 1369.396,A 0.000,B 0.000,C 90.000,E1 107.221} C_DIS
LIN {X 0.287,Y -661.116,Z 1369.393,A 0.000,B 0.000,C 90.000,E1 106.677} C_DIS
LIN {X 0.089,Y -662.926,Z 1369.390,A 0.000,B 0.000,C 90.000,E1 106.205} C_DIS
LIN {X 0.084,Y -664.531,Z 1369.387,A 0.000,B 0.000,C 90.000,E1 105.717} C_DIS
LIN {X -0.178,Y -666.367,Z 1369.383,A 0.000,B 0.000,C 90.000,E1 105.009} C_DIS
LIN {X -0.340,Y -667.341,Z 1369.381,A 0.000,B 0.000,C 90.000,E1 104.537} C_DIS
LIN {X 0.078,Y -668.370,Z 1369.377,A 0.000,B 0.000,C 90.000,E1 103.772} C_DIS
LIN {X -0.069,Y -668.827,Z 1369.374,A 0.000,B 0.000,C 90.000,E1 103.300} C_DIS
LIN {X -0.285,Y -669.033,Z 1369.370,A 0.000,B 0.000,C 90.000,E1 102.591} C_DIS
LIN {X 0.223,Y -668.988,Z 1369.367,A 0.000,B 0.000,C 90.000,E1 102.063} C_DIS
LIN {X 0.075,Y -668.771,Z 1369.365,A 0.000,B 0.000,C 90.000,E1 101.591} C_DIS
LIN {X -0.283,Y -667.923,Z 1369.360,A 0.000,B 0.000,C 90.000,E1 100.894} C_DIS
LIN {X 0.214,Y -667.181,Z 1369.358,A 0.000,B 0.000,C 90.000,E1 100.366} C_DIS
LIN {X -0.069,Y -666.211,Z 1369.355,A 0.000,B 0.000,C 90.000,E1 99.905} C_DIS
LIN {X -0.244,Y -664.959,Z 1369.352,A 0.000,B 0.000,C 90.000,E1 99.434} C_DIS
LIN {X 0.118,Y -663.541,Z 1369.350,A 0.000,B 0.000,C 90.000,E1 98.916} C_DIS
LIN {X -0.283,Y -660.933,Z 1369.346,A 0.000,B 0.000,C 90.000,E1 98.219} C_DIS
LIN {X 0.058,Y -659.040,Z 1369.343,A 0.000,B 0.000,C 90.000,E1 97.701} C_DIS
LIN {X 0.051,Y -654.529,Z 1369.337,A 0.000,B 0.000,C 90.000,E1 96.720} C_DIS
LIN {X 0.241,Y -651.153,Z 1369.334,A 0.000,B 0.000,C 90.000,E1 96.087} C_DIS
LIN {X -0.243,Y -647.497,Z 1369.331,A 0.000,B 0.000,C 90.000,E1 95.511} C_DIS
LIN {X -0.111,Y -643.590,Z 1369.327,A 0.000,B 0.000,C 90.000,E1 94.878} C_DIS
LIN {X -0.013,Y -639.516,Z 1369.324,A 0.000,B 0.000,C 90.000,E1 94.245} C_DIS
LIN {X 0.298,Y -636.846,Z 1369.322,A 0.000,B 0.000,C 90.000,E1 93.841} C_DIS
LIN {X -0.209,Y -632.906,Z 1369.319,A 0.000,B 0.000,C 90.000,E1 93.383} C_DIS
LIN {X -0.072,Y -628.451,Z 1369.316,A 0.000,B 0.000,C 90.000,E1 92.865} C_DIS
LIN {X -0.005,Y -622.239,Z 1369.313,A 0.000,B 0.000,C 90.000,E1 92.236} C_DIS
LIN {X 0.154,Y -615.862,Z 1369.309,A 0.000,B 0.000,C 90.000,E1 91.604} C_DIS
LIN {X -0.124,Y -610.540,Z 1369.306,A 0.000,B 0.000,C 90.000,E1 91.146} C_DIS
LIN {X -0.035,Y -603.251,Z 1369.303,A 0.000,B 0.000,C 90.000,E1 90.573} C_DIS
LIN {X -0.090,Y -596.569,Z 1369.301,A 0.000,B 0.000,C 90.000,E1 90.172} C_DIS
LIN {X -0.121,Y -589.690,Z 1369.299,A 0.000,B 0.000,C 90.000,E1 89.828} C_DIS
LIN {X -0.242,Y -582.583,Z 1369.297,A 0.000,B 0.000,C 90.000,E1 89.542} C_DIS
LIN {X 0.101,Y -578.446,Z 1369.296,A 0.000,B 0.000,C 90.000,E1 89.312} C_DIS
LIN {X 0.281,Y -576.488,Z 1369.295,A 0.000,B 0.000,C 90.000,E1 89.141} C_DIS
LIN {X 0.137,Y -574.341,Z 1369.294,A 0.000,B 0.000,C 90.000,E1 88.969} C_DIS
LIN {X 0.100,Y -574.314,Z 1369.294,A 0.000,B 0.000,C 90.000,E1 88.969} C_DIS
LIN {X -0.132,Y -573.582,Z 1369.293,A 0.000,B 0.000,C 90.000,E1 88.740} C_DIS
LIN {X 0.062,Y -573.721,Z 1369.290,A 0.000,B 0.000,C 90.000,E1 88.108} C_DIS
LIN {X 0.126,Y -575.516,Z 1369.277,A 0.000,B 0.000,C 90.000,E1 85.927} C_DIS
LIN {X -0.157,Y -578.036,Z 1369.264,A 0.000,B 0.000,C 90.000,E1 83.514} C_DIS
LIN {X -0.180,Y -580.014,Z 1369.255,A 0.000,B 0.000,C 90.000,E1 81.894} C_DIS
LIN {X -0.162,Y -581.947,Z 1369.246,A 0.000,B 0.000,C 90.000,E1 80.274} C_DIS
LIN {X 0.198,Y -583.180,Z 1369.240,A 0.000,B 0.000,C 90.000,E1 79.162} C_DIS
LIN {X -0.201,Y -584.773,Z 1369.231,A 0.000,B 0.000,C 90.000,E1 77.589} C_DIS
LIN {X 0.009,Y -585.936,Z 1369.224,A 0.000,B 0.000,C 90.000,E1 76.228} C_DIS
LIN {X -0.073,Y -587.108,Z 1369.215,A 0.000,B 0.000,C 90.000,E1 74.629} C_DIS
LIN {X 0.178,Y -587.946,Z 1369.207,A 0.000,B 0.000,C 90.000,E1 73.268} C_DIS
LIN {X 0.044,Y -588.820,Z 1369.200,A 0.000,B 0.000,C 90.000,E1 71.945} C_DIS
LIN {X 0.219,Y -589.831,Z 1369.189,A 0.000,B 0.000,C 90.000,E1 70.061} C_DIS
LIN {X -0.242,Y -590.624,Z 1369.182,A 0.000,B 0.000,C 90.000,E1 68.773} C_DIS
LIN {X -0.256,Y -591.649,Z 1369.173,A 0.000,B 0.000,C 90.000,E1 67.177} C_DIS
LIN {X 0.313,Y -592.684,Z 1369.166,A 0.000,B 0.000,C 90.000,E1 65.793} C_DIS
LIN {X 0.113,Y -593.836,Z 1369.158,A 0.000,B 0.000,C 90.000,E1 64.485} C_DIS
LIN {X -0.178,Y -594.990,Z 1369.150,A 0.000,B 0.000,C 90.000,E1 62.922} C_DIS
LIN {X -0.074,Y -596.719,Z 1369.138,A 0.000,B 0.000,C 90.000,E1 60.795} C_DIS
LIN {X 0.087,Y -597.924,Z 1369.130,A 0.000,B 0.000,C 90.000,E1 59.459} C_DIS
LIN {X 0.097,Y -599.767,Z 1369.120,A 0.000,B 0.000,C 90.000,E1 57.612} C_DIS
LIN {X -0.225,Y -601.465,Z 1369.110,A 0.000,B 0.000,C 90.000,E1 55.801} C_DIS
LIN {X 0.090,Y -602.931,Z 1369.101,A 0.000,B 0.000,C 90.000,E1 54.196} C_DIS
LIN {X 0.201,Y -604.598,Z 1369.091,A 0.000,B 0.000,C 90.000,E1 52.351} C_DIS
LIN {X -0.081,Y -605.377,Z 1369.085,A 0.000,B 0.000,C 90.000,E1 51.331} C_DIS
LIN {X 0.092,Y -606.197,Z 1369.076,A 0.000,B 0.000,C 90.000,E1 49.747} C_DIS
LIN {X 0.221,Y -606.720,Z 1369.071,A 0.000,B 0.000,C 90.000,E1 48.690} C_DIS
LIN {X -0.096,Y -607.048,Z 1369.065,A 0.000,B 0.000,C 90.000,E1 47.676} C_DIS
LIN {X -0.155,Y -607.294,Z 1369.058,A 0.000,B 0.000,C 90.000,E1 46.377} C_DIS
LIN {X 0.140,Y -607.326,Z 1369.053,A 0.000,B 0.000,C 90.000,E1 45.567} C_DIS
LIN {X 0.249,Y -607.244,Z 1369.047,A 0.000,B 0.000,C 90.000,E1 44.514} C_DIS
LIN {X -0.064,Y -606.962,Z 1369.042,A 0.000,B 0.000,C 90.000,E1 43.500} C_DIS
LIN {X -0.159,Y -606.339,Z 1369.034,A 0.000,B 0.000,C 90.000,E1 42.204} C_DIS
LIN {X -0.235,Y -605.686,Z 1369.027,A 0.000,B 0.000,C 90.000,E1 40.906} C_DIS
LIN {X 0.139,Y -604.834,Z 1369.020,A 0.000,B 0.000,C 90.000,E1 39.564} C_DIS
LIN {X -0.139,Y -604.033,Z 1369.014,A 0.000,B 0.000,C 90.000,E1 38.543} C_DIS
LIN {X -0.169,Y -602.828,Z 1369.007,A 0.000,B 0.000,C 90.000,E1 37.237} C_DIS
LIN {X 0.010,Y -601.659,Z 1369.001,A 0.000,B 0.000,C 90.000,E1 36.171} C_DIS
LIN {X -0.080,Y -599.527,Z 1368.994,A 0.000,B 0.000,C 90.000,E1 34.865} C_DIS
LIN {X -0.403,Y -596.744,Z 1368.986,A 0.000,B 0.000,C 90.000,E1 33.579} C_DIS
LIN {X 0.165,Y -594.168,Z 1368.980,A 0.000,B 0.000,C 90.000,E1 32.467} C_DIS
LIN {X 0.166,Y -591.940,Z 1368.976,A 0.000,B 0.000,C 90.000,E1 31.671} C_DIS
LIN {X 0.260,Y -590.337,Z 1368.973,A 0.000,B 0.000,C 90.000,E1 31.131} C_DIS
LIN {X 0.286,Y -585.511,Z 1368.966,A 0.000,B 0.000,C 90.000,E1 29.795} C_DIS
LIN {X 0.041,Y -583.366,Z 1368.963,A 0.000,B 0.000,C 90.000,E1 29.283} C_DIS
LIN {X -0.065,Y -579.703,Z 1368.958,A 0.000,B 0.000,C 90.000,E1 28.487} C_DIS
LIN {X 0.364,Y -576.387,Z 1368.954,A 0.000,B 0.000,C 90.000,E1 27.769} C_DIS
LIN {X -0.094,Y -572.076,Z 1368.950,A 0.000,B 0.000,C 90.000,E1 27.001} C_DIS
LIN {X 0.006,Y -568.232,Z 1368.946,A 0.000,B 0.000,C 90.000,E1 26.309} C_DIS
LIN {X -0.096,Y -564.923,Z 1368.943,A 0.000,B 0.000,C 90.000,E1 25.771} C_DIS
LIN {X 0.037,Y -561.401,Z 1368.940,A 0.000,B 0.000,C 90.000,E1 25.207} C_DIS
LIN {X 0.041,Y -556.682,Z 1368.936,A 0.000,B 0.000,C 90.000,E1 24.515} C_DIS
LIN {X -0.108,Y -550.662,Z 1368.932,A 0.000,B 0.000,C 90.000,E1 23.695} C_DIS
LIN {X 0.305,Y -545.161,Z 1368.928,A 0.000,B 0.000,C 90.000,E1 22.950} C_DIS
LIN {X 0.088,Y -540.484,Z 1368.925,A 0.000,B 0.000,C 90.000,E1 22.408} C_DIS
LIN {X -0.090,Y -534.337,Z 1368.921,A 0.000,B 0.000,C 90.000,E1 21.716} C_DIS
LIN {X 0.171,Y -523.994,Z 1368.914,A 0.000,B 0.000,C 90.000,E1 20.556} C_DIS
LIN {X -0.007,Y -511.946,Z 1368.907,A 0.000,B 0.000,C 90.000,E1 19.322} C_DIS
LIN {X 0.245,Y -503.052,Z 1368.902,A 0.000,B 0.000,C 90.000,E1 18.362} C_DIS
LIN {X 0.178,Y -492.241,Z 1368.896,A 0.000,B 0.000,C 90.000,E1 17.275} C_DIS
LIN {X 0.151,Y -478.233,Z 1368.888,A 0.000,B 0.000,C 90.000,E1 15.898} C_DIS
LIN {X 0.193,Y -464.222,Z 1368.881,A 0.000,B 0.000,C 90.000,E1 14.481} C_DIS
LIN {X 0.024,Y -452.769,Z 1368.874,A 0.000,B 0.000,C 90.000,E1 13.355} C_DIS
LIN {X 0.035,Y -438.646,Z 1368.866,A 0.000,B 0.000,C 90.000,E1 11.883} C_DIS
LIN {X 0.013,Y -429.039,Z 1368.860,A 0.000,B 0.000,C 90.000,E1 10.838} C_DIS
LIN {X -0.120,Y -415.094,Z 1368.851,A 0.000,B 0.000,C 90.000,E1 9.265} C_DIS
LIN {X 0.074,Y -402.403,Z 1368.843,A 0.000,B 0.000,C 90.000,E1 7.757} C_DIS
LIN {X -0.090,Y -396.770,Z 1368.840,A 0.000,B 0.000,C 90.000,E1 7.125} C_DIS
LIN {X 0.144,Y -392.674,Z 1368.836,A 0.000,B 0.000,C 90.000,E1 6.486} C_DIS
LIN {X 0.117,Y -392.450,Z 1368.836,A 0.000,B 0.000,C 90.000,E1 6.429} C_DIS
LIN {X 0.080,Y -392.444,Z 1368.836,A 0.000,B 0.000,C 90.000,E1 6.429} C_DIS
LIN {X 0.103,Y -393.077,Z 1368.835,A 0.000,B 0.000,C 90.000,E1 6.315} C_DIS
LIN {X 0.060,Y -394.309,Z 1368.834,A 0.000,B 0.000,C 90.000,E1 6.144} C_DIS
LIN {X 0.074,Y -398.891,Z 1368.832,A 0.000,B 0.000,C 90.000,E1 5.739} C_DIS
LIN {X -0.106,Y -405.767,Z 1368.829,A 0.000,B 0.000,C 90.000,E1 5.277} C_DIS
LIN {X 0.058,Y -411.920,Z 1368.827,A 0.000,B 0.000,C 90.000,E1 4.759} C_DIS
LIN {X 0.006,Y -417.963,Z 1368.824,A 0.000,B 0.000,C 90.000,E1 4.245} C_DIS
LIN {X 0.020,Y -423.627,Z 1368.820,A 0.000,B 0.000,C 90.000,E1 3.669} C_DIS
LIN {X 0.119,Y -430.453,Z 1368.816,A 0.000,B 0.000,C 90.000,E1 2.865} C_DIS
LIN {X -0.118,Y -435.704,Z 1368.812,A 0.000,B 0.000,C 90.000,E1 2.236} C_DIS
LIN {X 0.149,Y -442.017,Z 1368.808,A 0.000,B 0.000,C 90.000,E1 1.375} C_DIS
LIN {X -0.046,Y -446.808,Z 1368.804,A 0.000,B 0.000,C 90.000,E1 0.745} C_DIS
LIN {X 0.000,Y -452.014,Z 1368.800,A 0.000,B 0.000,C 90.000,E1 360.000} C_DIS
LIN {X 0.063,Y -457.568,Z 1368.795,A 0.000,B 0.000,C 90.000,E1 359.141} C_DIS
LIN {X -0.016,Y -461.590,Z 1368.792,A 0.000,B 0.000,C 90.000,E1 358.511} C_DIS
LIN {X 0.060,Y -466.165,Z 1368.787,A 0.000,B 0.000,C 90.000,E1 357.707} C_DIS
LIN {X 0.160,Y -470.491,Z 1368.783,A 0.000,B 0.000,C 90.000,E1 356.906} C_DIS
LIN {X -0.146,Y -474.433,Z 1368.779,A 0.000,B 0.000,C 90.000,E1 356.159} C_DIS
LIN {X 0.057,Y -478.071,Z 1368.774,A 0.000,B 0.000,C 90.000,E1 355.355} C_DIS
LIN {X -0.182,Y -481.382,Z 1368.770,A 0.000,B 0.000,C 90.000,E1 354.609} C_DIS
LIN {X 0.137,Y -484.434,Z 1368.766,A 0.000,B 0.000,C 90.000,E1 353.799} C_DIS
LIN {X 0.155,Y -487.778,Z 1368.761,A 0.000,B 0.000,C 90.000,E1 352.875} C_DIS
LIN {X 0.209,Y -490.807,Z 1368.755,A 0.000,B 0.000,C 90.000,E1 351.951} C_DIS
LIN {X -0.192,Y -493.436,Z 1368.750,A 0.000,B 0.000,C 90.000,E1 351.084} C_DIS
LIN {X -0.001,Y -495.746,Z 1368.745,A 0.000,B 0.000,C 90.000,E1 350.151} C_DIS
LIN {X 0.223,Y -497.873,Z 1368.740,A 0.000,B 0.000,C 90.000,E1 349.218} C_DIS
LIN {X -0.094,Y -500.347,Z 1368.734,A 0.000,B 0.000,C 90.000,E1 348.049} C_DIS
LIN {X 0.108,Y -502.445,Z 1368.727,A 0.000,B 0.000,C 90.000,E1 346.825} C_DIS
LIN {X 0.038,Y -502.948,Z 1368.725,A 0.000,B 0.000,C 90.000,E1 346.533} C_DIS
LIN {X 0.090,Y -503.320,Z 1368.724,A 0.000,B 0.000,C 90.000,E1 346.228} C_DIS
LIN {X 0.023,Y -503.516,Z 1368.722,A 0.000,B 0.000,C 90.000,E1 345.936} C_DIS
LIN {X -0.041,Y -503.520,Z 1368.720,A 0.000,B 0.000,C 90.000,E1 345.644} C_DIS
LIN {X 0.020,Y -503.196,Z 1368.719,A 0.000,B 0.000,C 90.000,E1 345.338} C_DIS
LIN {X -0.045,Y -502.281,Z 1368.717,A 0.000,B 0.000,C 90.000,E1 345.046} C_DIS
LIN {X 0.228,Y -501.252,Z 1368.716,A 0.000,B 0.000,C 90.000,E1 344.866} C_DIS
LIN {X 0.059,Y -499.936,Z 1368.716,A 0.000,B 0.000,C 90.000,E1 344.810} C_DIS
LIN {X 0.137,Y -465.999,Z 1368.709,A 0.000,B 0.000,C 90.000,E1 343.685} C_DIS
LIN {X -0.214,Y -434.711,Z 1368.703,A 0.000,B 0.000,C 90.000,E1 342.543} C_DIS
LIN {X -0.123,Y -407.107,Z 1368.696,A 0.000,B 0.000,C 90.000,E1 341.329} C_DIS
LIN {X 0.048,Y -383.147,Z 1368.690,A 0.000,B 0.000,C 90.000,E1 340.115} C_DIS
LIN {X -0.134,Y -361.971,Z 1368.683,A 0.000,B 0.000,C 90.000,E1 338.954} C_DIS
LIN {X 0.184,Y -361.945,Z 1368.683,A 0.000,B 0.000,C 90.000,E1 338.901} C_DIS
LIN {X -0.050,Y -365.967,Z 1368.643,A 0.000,B 0.000,C 90.000,E1 331.691} C_DIS
LIN {X 0.112,Y -366.382,Z 1368.639,A 0.000,B 0.000,C 90.000,E1 330.923} C_DIS
LIN {X 0.054,Y -371.340,Z 1368.604,A 0.000,B 0.000,C 90.000,E1 324.642} C_DIS
LIN {X 0.041,Y -371.757,Z 1368.602,A 0.000,B 0.000,C 90.000,E1 324.276} C_DIS
LIN {X -0.183,Y -377.341,Z 1368.567,A 0.000,B 0.000,C 90.000,E1 318.081} C_DIS
LIN {X 0.097,Y -378.227,Z 1368.563,A 0.000,B 0.000,C 90.000,E1 317.310} C_DIS
LIN {X 0.088,Y -383.923,Z 1368.531,A 0.000,B 0.000,C 90.000,E1 311.515} C_DIS
LIN {X -0.118,Y -384.883,Z 1368.527,A 0.000,B 0.000,C 90.000,E1 310.825} C_DIS
LIN {X -0.197,Y -390.593,Z 1368.495,A 0.000,B 0.000,C 90.000,E1 305.105} C_DIS
LIN {X -0.129,Y -391.087,Z 1368.493,A 0.000,B 0.000,C 90.000,E1 304.739} C_DIS
LIN {X 0.108,Y -391.640,Z 1368.489,A 0.000,B 0.000,C 90.000,E1 303.992} C_DIS
LIN {X 0.007,Y -396.809,Z 1368.459,A 0.000,B 0.000,C 90.000,E1 298.693} C_DIS
LIN {X -0.124,Y -397.114,Z 1368.458,A 0.000,B 0.000,C 90.000,E1 298.359} C_DIS
LIN {X 0.033,Y -401.587,Z 1368.426,A 0.000,B 0.000,C 90.000,E1 292.717} C_DIS
LIN {X -0.077,Y -404.647,Z 1368.395,A 0.000,B 0.000,C 90.000,E1 287.149} C_DIS
LIN {X 0.008,Y -404.736,Z 1368.391,A 0.000,B 0.000,C 90.000,E1 286.441} C_DIS
LIN {X -0.096,Y -406.093,Z 1368.364,A 0.000,B 0.000,C 90.000,E1 281.591} C_DIS
LIN {X -0.088,Y -406.100,Z 1368.362,A 0.000,B 0.000,C 90.000,E1 281.243} C_DIS
LIN {X -0.052,Y -405.677,Z 1368.333,A 0.000,B 0.000,C 90.000,E1 276.030} C_DIS
LIN {X -0.044,Y -405.292,Z 1368.330,A 0.000,B 0.000,C 90.000,E1 275.334} C_DIS
LIN {X 0.028,Y -403.504,Z 1368.305,A 0.000,B 0.000,C 90.000,E1 270.802} C_DIS
LIN {X -0.005,Y -403.296,Z 1368.303,A 0.000,B 0.000,C 90.000,E1 270.458} C_DIS
LIN {X 0.177,Y -398.943,Z 1368.271,A 0.000,B 0.000,C 90.000,E1 264.837} C_DIS
LIN {X 0.046,Y -393.118,Z 1368.242,A 0.000,B 0.000,C 90.000,E1 259.567} C_DIS
LIN {X 0.007,Y -392.848,Z 1368.240,A 0.000,B 0.000,C 90.000,E1 259.218} C_DIS
LIN {X 0.120,Y -386.006,Z 1368.212,A 0.000,B 0.000,C 90.000,E1 254.212} C_DIS
LIN {X 0.060,Y -385.280,Z 1368.208,A 0.000,B 0.000,C 90.000,E1 253.504} C_DIS
LIN {X 0.082,Y -384.791,Z 1368.206,A 0.000,B 0.000,C 90.000,E1 253.142} C_DIS
LIN {X -0.046,Y -377.989,Z 1368.182,A 0.000,B 0.000,C 90.000,E1 248.827} C_DIS
LIN {X 0.040,Y -376.247,Z 1368.174,A 0.000,B 0.000,C 90.000,E1 247.358} C_DIS
LIN {X 0.141,Y -374.969,Z 1368.170,A 0.000,B 0.000,C 90.000,E1 246.613} C_DIS
LIN {X -0.124,Y -368.435,Z 1368.148,A 0.000,B 0.000,C 90.000,E1 242.615} C_DIS
LIN {X 0.181,Y -366.072,Z 1368.138,A 0.000,B 0.000,C 90.000,E1 240.717} C_DIS
LIN {X 0.088,Y -359.215,Z 1368.115,A 0.000,B 0.000,C 90.000,E1 236.628} C_DIS
LIN {X 0.105,Y -355.866,Z 1368.100,A 0.000,B 0.000,C 90.000,E1 233.989} C_DIS
LIN {X -0.091,Y -348.811,Z 1368.075,A 0.000,B 0.000,C 90.000,E1 229.461} C_DIS
LIN {X -0.015,Y -346.199,Z 1368.062,A 0.000,B 0.000,C 90.000,E1 227.148} C_DIS
LIN {X -0.006,Y -345.086,Z 1368.058,A 0.000,B 0.000,C 90.000,E1 226.377} C_DIS
LIN {X -0.078,Y -338.600,Z 1368.030,A 0.000,B 0.000,C 90.000,E1 221.353} C_DIS
LIN {X -0.086,Y -336.855,Z 1368.019,A 0.000,B 0.000,C 90.000,E1 219.402} C_DIS
LIN {X 0.096,Y -330.873,Z 1367.988,A 0.000,B 0.000,C 90.000,E1 213.865} C_DIS
LIN {X -0.051,Y -329.304,Z 1367.975,A 0.000,B 0.000,C 90.000,E1 211.514} C_DIS
LIN {X 0.015,Y -324.873,Z 1367.944,A 0.000,B 0.000,C 90.000,E1 205.924} C_DIS
LIN {X -0.128,Y -324.095,Z 1367.934,A 0.000,B 0.000,C 90.000,E1 204.079} C_DIS
LIN {X -0.145,Y -324.118,Z 1367.934,A 0.000,B 0.000,C 90.000,E1 204.079} C_DIS
LIN {X -0.064,Y -344.730,Z 1367.926,A 0.000,B 0.000,C 90.000,E1 202.589} C_DIS
LIN {X 0.056,Y -367.323,Z 1367.918,A 0.000,B 0.000,C 90.000,E1 201.153} C_DIS
LIN {X 0.027,Y -391.851,Z 1367.910,A 0.000,B 0.000,C 90.000,E1 199.812} C_DIS
LIN {X 0.021,Y -418.321,Z 1367.903,A 0.000,B 0.000,C 90.000,E1 198.544} C_DIS
LIN {X 0.186,Y -444.973,Z 1367.897,A 0.000,B 0.000,C 90.000,E1 197.402} C_DIS
LIN {X 0.084,Y -446.677,Z 1367.896,A 0.000,B 0.000,C 90.000,E1 197.275} C_DIS
LIN {X -0.062,Y -448.043,Z 1367.895,A 0.000,B 0.000,C 90.000,E1 197.040} C_DIS
LIN {X 0.228,Y -449.088,Z 1367.893,A 0.000,B 0.000,C 90.000,E1 196.677} C_DIS
LIN {X -0.036,Y -449.772,Z 1367.891,A 0.000,B 0.000,C 90.000,E1 196.386} C_DIS
LIN {X -0.168,Y -450.225,Z 1367.889,A 0.000,B 0.000,C 90.000,E1 196.079} C_DIS
LIN {X 0.181,Y -450.982,Z 1367.884,A 0.000,B 0.000,C 90.000,E1 195.064} C_DIS
LIN {X -0.063,Y -452.039,Z 1367.875,A 0.000,B 0.000,C 90.000,E1 193.480} C_DIS
LIN {X -0.038,Y -452.666,Z 1367.868,A 0.000,B 0.000,C 90.000,E1 192.187} C_DIS
LIN {X 0.200,Y -453.442,Z 1367.859,A 0.000,B 0.000,C 90.000,E1 190.546} C_DIS
LIN {X -0.061,Y -453.739,Z 1367.853,A 0.000,B 0.000,C 90.000,E1 189.613} C_DIS
LIN {X -0.203,Y -454.122,Z 1367.843,A 0.000,B 0.000,C 90.000,E1 187.701} C_DIS
LIN {X 0.135,Y -454.307,Z 1367.836,A 0.000,B 0.000,C 90.000,E1 186.372} C_DIS
LIN {X -0.025,Y -454.428,Z 1367.828,A 0.000,B 0.000,C 90.000,E1 185.106} C_DIS
LIN {X -0.016,Y -454.156,Z 1367.819,A 0.000,B 0.000,C 90.000,E1 183.498} C_DIS
LIN {X 0.072,Y -453.777,Z 1367.814,A 0.000,B 0.000,C 90.000,E1 182.522} C_DIS
LIN {X -0.130,Y -453.042,Z 1367.807,A 0.000,B 0.000,C 90.000,E1 181.260} C_DIS
LIN {X -0.070,Y -452.051,Z 1367.802,A 0.000,B 0.000,C 90.000,E1 180.286} C_DIS
LIN {X -0.187,Y -451.236,Z 1367.798,A 0.000,B 0.000,C 90.000,E1 179.656} C_DIS
LIN {X -0.149,Y -449.704,Z 1367.793,A 0.000,B 0.000,C 90.000,E1 178.682} C_DIS
LIN {X 0.179,Y -448.419,Z 1367.789,A 0.000,B 0.000,C 90.000,E1 177.993} C_DIS
LIN {X 0.176,Y -445.753,Z 1367.784,A 0.000,B 0.000,C 90.000,E1 177.020} C_DIS
LIN {X 0.032,Y -443.842,Z 1367.780,A 0.000,B 0.000,C 90.000,E1 176.388} C_DIS
LIN {X -0.064,Y -440.704,Z 1367.776,A 0.000,B 0.000,C 90.000,E1 175.584} C_DIS
LIN {X -0.193,Y -437.161,Z 1367.771,A 0.000,B 0.000,C 90.000,E1 174.780} C_DIS
LIN {X -0.056,Y -435.470,Z 1367.769,A 0.000,B 0.000,C 90.000,E1 174.432} C_DIS
LIN {X 0.156,Y -431.947,Z 1367.765,A 0.000,B 0.000,C 90.000,E1 173.742} C_DIS
LIN {X 0.010,Y -425.742,Z 1367.760,A 0.000,B 0.000,C 90.000,E1 172.761} C_DIS
LIN {X -0.207,Y -418.941,Z 1367.754,A 0.000,B 0.000,C 90.000,E1 171.781} C_DIS
LIN {X 0.085,Y -406.219,Z 1367.744,A 0.000,B 0.000,C 90.000,E1 169.859} C_DIS
LIN {X 0.098,Y -394.318,Z 1367.733,A 0.000,B 0.000,C 90.000,E1 167.937} C_DIS
LIN {X 0.104,Y -390.267,Z 1367.729,A 0.000,B 0.000,C 90.000,E1 167.229} C_DIS
LIN {X 0.081,Y -387.110,Z 1367.725,A 0.000,B 0.000,C 90.000,E1 166.520} C_DIS
LIN {X 0.138,Y -386.082,Z 1367.723,A 0.000,B 0.000,C 90.000,E1 166.172} C_DIS
LIN {X 0.220,Y -385.698,Z 1367.722,A 0.000,B 0.000,C 90.000,E1 165.992} C_DIS
LIN {X -0.167,Y -385.624,Z 1367.721,A 0.000,B 0.000,C 90.000,E1 165.880} C_DIS
LIN {X -0.030,Y -385.751,Z 1367.720,A 0.000,B 0.000,C 90.000,E1 165.644} C_DIS
LIN {X -0.068,Y -385.778,Z 1367.720,A 0.000,B 0.000,C 90.000,E1 165.644} C_DIS
LIN {X -0.047,Y -387.342,Z 1367.719,A 0.000,B 0.000,C 90.000,E1 165.338} C_DIS
LIN {X -0.135,Y -388.135,Z 1367.718,A 0.000,B 0.000,C 90.000,E1 165.172} C_DIS
LIN {X -0.018,Y -393.788,Z 1367.714,A 0.000,B 0.000,C 90.000,E1 164.448} C_DIS
LIN {X 0.171,Y -398.349,Z 1367.711,A 0.000,B 0.000,C 90.000,E1 163.921} C_DIS
LIN {X -0.101,Y -410.160,Z 1367.705,A 0.000,B 0.000,C 90.000,E1 162.834} C_DIS
LIN {X -0.038,Y -429.105,Z 1367.696,A 0.000,B 0.000,C 90.000,E1 161.221} C_DIS
LIN {X -0.134,Y -451.412,Z 1367.686,A 0.000,B 0.000,C 90.000,E1 159.518} C_DIS
LIN {X 0.010,Y -459.154,Z 1367.683,A 0.000,B 0.000,C 90.000,E1 158.901} C_DIS
LIN {X 0.077,Y -466.735,Z 1367.679,A 0.000,B 0.000,C 90.000,E1 158.284} C_DIS
LIN {X -0.008,Y -472.691,Z 1367.677,A 0.000,B 0.000,C 90.000,E1 157.794} C_DIS
LIN {X 0.124,Y -481.571,Z 1367.672,A 0.000,B 0.000,C 90.000,E1 156.997} C_DIS
LIN {X 0.150,Y -492.944,Z 1367.666,A 0.000,B 0.000,C 90.000,E1 155.921} C_DIS
LIN {X 0.248,Y -499.775,Z 1367.663,A 0.000,B 0.000,C 90.000,E1 155.229} C_DIS
LIN {X -0.178,Y -505.053,Z 1367.659,A 0.000,B 0.000,C 90.000,E1 154.717} C_DIS
LIN {X -0.130,Y -514.015,Z 1367.654,A 0.000,B 0.000,C 90.000,E1 153.691} C_DIS
LIN {X 0.100,Y -518.837,Z 1367.651,A 0.000,B 0.000,C 90.000,E1 153.076} C_DIS
LIN {X -0.024,Y -524.317,Z 1367.646,A 0.000,B 0.000,C 90.000,E1 152.359} C_DIS
LIN {X -0.098,Y -526.456,Z 1367.645,A 0.000,B 0.000,C 90.000,E1 152.076} C_DIS
LIN {X -0.251,Y -530.192,Z 1367.642,A 0.000,B 0.000,C 90.000,E1 151.513} C_DIS
LIN {X -0.276,Y -534.061,Z 1367.638,A 0.000,B 0.000,C 90.000,E1 150.795} C_DIS
LIN {X -0.125,Y -536.712,Z 1367.634,A 0.000,B 0.000,C 90.000,E1 150.205} C_DIS
LIN {X 0.040,Y -540.112,Z 1367.630,A 0.000,B 0.000,C 90.000,E1 149.331} C_DIS
LIN {X 0.233,Y -542.141,Z 1367.627,A 0.000,B 0.000,C 90.000,E1 148.742} C_DIS
LIN {X -0.024,Y -543.861,Z 1367.623,A 0.000,B 0.000,C 90.000,E1 148.201} C_DIS
LIN {X 0.220,Y -546.070,Z 1367.619,A 0.000,B 0.000,C 90.000,E1 147.327} C_DIS
LIN {X -0.012,Y -547.336,Z 1367.615,A 0.000,B 0.000,C 90.000,E1 146.786} C_DIS
LIN {X -0.147,Y -549.332,Z 1367.609,A 0.000,B 0.000,C 90.000,E1 145.674} C_DIS
LIN {X 0.009,Y -550.621,Z 1367.605,A 0.000,B 0.000,C 90.000,E1 144.815} C_DIS
LIN {X -0.137,Y -551.680,Z 1367.600,A 0.000,B 0.000,C 90.000,E1 143.989} C_DIS
LIN {X 0.112,Y -552.751,Z 1367.594,A 0.000,B 0.000,C 90.000,E1 142.844} C_DIS
LIN {X -0.057,Y -553.619,Z 1367.588,A 0.000,B 0.000,C 90.000,E1 141.743} C_DIS
LIN {X -0.076,Y -554.700,Z 1367.578,A 0.000,B 0.000,C 90.000,E1 140.070} C_DIS
LIN {X -0.150,Y -555.699,Z 1367.569,A 0.000,B 0.000,C 90.000,E1 138.405} C_DIS
LIN {X 0.165,Y -556.527,Z 1367.560,A 0.000,B 0.000,C 90.000,E1 136.701} C_DIS
LIN {X -0.308,Y -557.178,Z 1367.550,A 0.000,B 0.000,C 90.000,E1 135.081} C_DIS
LIN {X 0.089,Y -557.951,Z 1367.540,A 0.000,B 0.000,C 90.000,E1 133.095} C_DIS
LIN {X -0.137,Y -559.309,Z 1367.526,A 0.000,B 0.000,C 90.000,E1 130.620} C_DIS
LIN {X 0.172,Y -559.921,Z 1367.523,A 0.000,B 0.000,C 90.000,E1 130.172} C_DIS
LIN {X -0.219,Y -561.401,Z 1367.521,A 0.000,B 0.000,C 90.000,E1 129.806} C_DIS
LIN {X 0.098,Y -561.432,Z 1367.521,A 0.000,B 0.000,C 90.000,E1 129.769} C_DIS
LIN {X 0.312,Y -563.076,Z 1367.521,A 0.000,B 0.000,C 90.000,E1 129.644} C_DIS
LIN {X -0.005,Y -568.589,Z 1367.519,A 0.000,B 0.000,C 90.000,E1 129.483} C_DIS
LIN {X 0.060,Y -575.783,Z 1367.518,A 0.000,B 0.000,C 90.000,E1 129.277} C_DIS
LIN {X -0.073,Y -578.739,Z 1367.518,A 0.000,B 0.000,C 90.000,E1 129.197} C_DIS
LIN {X 0.065,Y -581.802,Z 1367.517,A 0.000,B 0.000,C 90.000,E1 129.072} C_DIS
LIN {X 0.071,Y -587.476,Z 1367.516,A 0.000,B 0.000,C 90.000,E1 128.785} C_DIS
LIN {X -0.018,Y -590.509,Z 1367.515,A 0.000,B 0.000,C 90.000,E1 128.624} C_DIS
LIN {X -0.065,Y -596.256,Z 1367.513,A 0.000,B 0.000,C 90.000,E1 128.257} C_DIS
LIN {X 0.250,Y -601.873,Z 1367.510,A 0.000,B 0.000,C 90.000,E1 127.810} C_DIS
LIN {X -0.157,Y -608.648,Z 1367.507,A 0.000,B 0.000,C 90.000,E1 127.282} C_DIS
LIN {X -0.330,Y -612.673,Z 1367.505,A 0.000,B 0.000,C 90.000,E1 126.950} C_DIS
LIN {X -0.345,Y -621.327,Z 1367.500,A 0.000,B 0.000,C 90.000,E1 126.091} C_DIS
LIN {X -0.109,Y -627.296,Z 1367.497,A 0.000,B 0.000,C 90.000,E1 125.438} C_DIS
LIN {X 0.228,Y -631.790,Z 1367.494,A 0.000,B 0.000,C 90.000,E1 124.898} C_DIS
LIN {X 0.075,Y -634.988,Z 1367.492,A 0.000,B 0.000,C 90.000,E1 124.532} C_DIS
LIN {X -0.307,Y -641.870,Z 1367.487,A 0.000,B 0.000,C 90.000,E1 123.706} C_DIS
LIN {X 0.173,Y -646.358,Z 1367.484,A 0.000,B 0.000,C 90.000,E1 123.038} C_DIS
LIN {X 0.152,Y -650.543,Z 1367.480,A 0.000,B 0.000,C 90.000,E1 122.418} C_DIS
LIN {X 0.117,Y -653.646,Z 1367.477,A 0.000,B 0.000,C 90.000,E1 121.926} C_DIS
LIN {X -0.048,Y -657.028,Z 1367.474,A 0.000,B 0.000,C 90.000,E1 121.337} C_DIS
LIN {X 0.007,Y -660.041,Z 1367.471,A 0.000,B 0.000,C 90.000,E1 120.718} C_DIS
LIN {X 0.252,Y -662.124,Z 1367.468,A 0.000,B 0.000,C 90.000,E1 120.207} C_DIS
LIN {X 0.081,Y -664.766,Z 1367.464,A 0.000,B 0.000,C 90.000,E1 119.489} C_DIS
LIN {X 0.112,Y -666.137,Z 1367.461,A 0.000,B 0.000,C 90.000,E1 118.999} C_DIS
LIN {X 0.409,Y -667.372,Z 1367.458,A 0.000,B 0.000,C 90.000,E1 118.487} C_DIS
LIN {X 0.286,Y -668.370,Z 1367.454,A 0.000,B 0.000,C 90.000,E1 117.769} C_DIS
LIN {X -0.136,Y -668.585,Z 1367.450,A 0.000,B 0.000,C 90.000,E1 117.078} C_DIS
LIN {X 0.187,Y -668.554,Z 1367.448,A 0.000,B 0.000,C 90.000,E1 116.565} C_DIS
LIN {X 0.071,Y -668.100,Z 1367.444,A 0.000,B 0.000,C 90.000,E1 115.848} C_DIS
LIN {X 0.388,Y -667.648,Z 1367.441,A 0.000,B 0.000,C 90.000,E1 115.335} C_DIS
LIN {X -0.186,Y -667.032,Z 1367.438,A 0.000,B 0.000,C 90.000,E1 114.899} C_DIS
LIN {X 0.121,Y -665.868,Z 1367.436,A 0.000,B 0.000,C 90.000,E1 114.387} C_DIS
LIN {X -0.001,Y -665.133,Z 1367.434,A 0.000,B 0.000,C 90.000,E1 114.155} C_DIS
LIN {X 0.290,Y -662.297,Z 1367.432,A 0.000,B 0.000,C 90.000,E1 113.643} C_DIS
LIN {X 0.358,Y -661.468,Z 1367.431,A 0.000,B 0.000,C 90.000,E1 113.515} C_DIS
LIN {X -0.180,Y -660.158,Z 1367.430,A 0.000,B 0.000,C 90.000,E1 113.439} C_DIS
LIN {X 0.258,Y -654.477,Z 1367.428,A 0.000,B 0.000,C 90.000,E1 112.950} C_DIS
LIN {X -0.077,Y -649.680,Z 1367.427,A 0.000,B 0.000,C 90.000,E1 112.770} C_DIS
LIN {X 0.240,Y -643.512,Z 1367.425,A 0.000,B 0.000,C 90.000,E1 112.514} C_DIS
LIN {X -0.157,Y -635.158,Z 1367.424,A 0.000,B 0.000,C 90.000,E1 112.333} C_DIS
LIN {X -0.159,Y -628.082,Z 1367.423,A 0.000,B 0.000,C 90.000,E1 112.153} C_DIS
LIN {X -0.223,Y -628.067,Z 1367.423,A 0.000,B 0.000,C 90.000,E1 112.153} C_DIS
LIN {X -0.219,Y -628.563,Z 1367.423,A 0.000,B 0.000,C 90.000,E1 112.078} C_DIS
LIN {X -0.013,Y -637.068,Z 1367.417,A 0.000,B 0.000,C 90.000,E1 111.099} C_DIS
LIN {X 0.273,Y -641.978,Z 1367.414,A 0.000,B 0.000,C 90.000,E1 110.482} C_DIS
LIN {X 0.122,Y -644.641,Z 1367.412,A 0.000,B 0.000,C 90.000,E1 110.120} C_DIS
LIN {X 0.020,Y -647.897,Z 1367.409,A 0.000,B 0.000,C 90.000,E1 109.631} C_DIS
LIN {X -0.206,Y -652.015,Z 1367.405,A 0.000,B 0.000,C 90.000,E1 108.906} C_DIS
LIN {X 0.147,Y -657.242,Z 1367.399,A 0.000,B 0.000,C 90.000,E1 107.764} C_DIS
LIN {X 0.007,Y -660.463,Z 1367.395,A 0.000,B 0.000,C 90.000,E1 107.040} C_DIS
LIN {X -0.108,Y -663.287,Z 1367.391,A 0.000,B 0.000,C 90.000,E1 106.315} C_DIS
LIN {X 0.258,Y -665.593,Z 1367.387,A 0.000,B 0.000,C 90.000,E1 105.552} C_DIS
LIN {X 0.268,Y -666.864,Z 1367.384,A 0.000,B 0.000,C 90.000,E1 105.064} C_DIS
LIN {X 0.030,Y -668.273,Z 1367.380,A 0.000,B 0.000,C 90.000,E1 104.356} C_DIS
LIN {X -0.119,Y -668.997,Z 1367.377,A 0.000,B 0.000,C 90.000,E1 103.883} C_DIS
LIN {X 0.315,Y -669.603,Z 1367.373,A 0.000,B 0.000,C 90.000,E1 103.119} C_DIS
LIN {X 0.174,Y -669.772,Z 1367.370,A 0.000,B 0.000,C 90.000,E1 102.647} C_DIS
LIN {X -0.110,Y -669.764,Z 1367.368,A 0.000,B 0.000,C 90.000,E1 102.187} C_DIS
LIN {X -0.250,Y -669.557,Z 1367.365,A 0.000,B 0.000,C 90.000,E1 101.715} C_DIS
LIN {X 0.188,Y -668.825,Z 1367.361,A 0.000,B 0.000,C 90.000,E1 100.950} C_DIS
LIN {X -0.088,Y -668.164,Z 1367.358,A 0.000,B 0.000,C 90.000,E1 100.489} C_DIS
LIN {X -0.246,Y -667.222,Z 1367.356,A 0.000,B 0.000,C 90.000,E1 100.018} C_DIS
LIN {X 0.042,Y -665.323,Z 1367.352,A 0.000,B 0.000,C 90.000,E1 99.265} C_DIS
LIN {X -0.245,Y -663.841,Z 1367.349,A 0.000,B 0.000,C 90.000,E1 98.803} C_DIS
LIN {X 0.213,Y -662.078,Z 1367.346,A 0.000,B 0.000,C 90.000,E1 98.276} C_DIS
LIN {X -0.094,Y -660.186,Z 1367.343,A 0.000,B 0.000,C 90.000,E1 97.814} C_DIS
LIN {X 0.038,Y -656.888,Z 1367.339,A 0.000,B 0.000,C 90.000,E1 97.068} C_DIS
LIN {X -0.294,Y -654.513,Z 1367.337,A 0.000,B 0.000,C 90.000,E1 96.606} C_DIS
LIN {X 0.007,Y -651.833,Z 1367.334,A 0.000,B 0.000,C 90.000,E1 96.087} C_DIS
LIN {X 0.123,Y -647.364,Z 1367.330,A 0.000,B 0.000,C 90.000,E1 95.334} C_DIS
LIN {X 0.129,Y -642.629,Z 1367.326,A 0.000,B 0.000,C 90.000,E1 94.588} C_DIS
LIN {X 0.211,Y -638.410,Z 1367.322,A 0.000,B 0.000,C 90.000,E1 93.955} C_DIS
LIN {X -0.289,Y -634.571,Z 1367.319,A 0.000,B 0.000,C 90.000,E1 93.498} C_DIS
LIN {X -0.272,Y -629.031,Z 1367.316,A 0.000,B 0.000,C 90.000,E1 92.865} C_DIS
LIN {X -0.113,Y -622.949,Z 1367.312,A 0.000,B 0.000,C 90.000,E1 92.236} C_DIS
LIN {X 0.029,Y -616.564,Z 1367.309,A 0.000,B 0.000,C 90.000,E1 91.604} C_DIS
LIN {X -0.271,Y -611.237,Z 1367.306,A 0.000,B 0.000,C 90.000,E1 91.146} C_DIS
LIN {X 0.237,Y -608.294,Z 1367.305,A 0.000,B 0.000,C 90.000,E1 90.859} C_DIS
LIN {X -0.153,Y -602.423,Z 1367.302,A 0.000,B 0.000,C 90.000,E1 90.458} C_DIS
LIN {X 0.294,Y -597.273,Z 1367.301,A 0.000,B 0.000,C 90.000,E1 90.115} C_DIS
LIN {X 0.191,Y -593.788,Z 1367.300,A 0.000,B 0.000,C 90.000,E1 89.943} C_DIS
LIN {X -0.058,Y -588.458,Z 1367.298,A 0.000,B 0.000,C 90.000,E1 89.714} C_DIS
LIN {X -0.068,Y -581.649,Z 1367.297,A 0.000,B 0.000,C 90.000,E1 89.427} C_DIS
LIN {X -0.060,Y -578.083,Z 1367.296,A 0.000,B 0.000,C 90.000,E1 89.255} C_DIS
LIN {X 0.191,Y -574.295,Z 1367.294,A 0.000,B 0.000,C 90.000,E1 88.912} C_DIS
LIN {X 0.153,Y -574.258,Z 1367.294,A 0.000,B 0.000,C 90.000,E1 88.912} C_DIS
LIN {X 0.070,Y -573.571,Z 1367.293,A 0.000,B 0.000,C 90.000,E1 88.682} C_DIS
LIN {X 0.265,Y -573.684,Z 1367.289,A 0.000,B 0.000,C 90.000,E1 88.051} C_DIS
LIN {X 0.037,Y -575.978,Z 1367.274,A 0.000,B 0.000,C 90.000,E1 85.355} C_DIS
LIN {X 0.247,Y -578.312,Z 1367.262,A 0.000,B 0.000,C 90.000,E1 83.166} C_DIS
LIN {X 0.015,Y -579.992,Z 1367.255,A 0.000,B 0.000,C 90.000,E1 81.837} C_DIS
LIN {X 0.130,Y -581.918,Z 1367.246,A 0.000,B 0.000,C 90.000,E1 80.208} C_DIS
LIN {X -0.184,Y -583.142,Z 1367.240,A 0.000,B 0.000,C 90.000,E1 79.162} C_DIS
LIN {X 0.113,Y -584.720,Z 1367.231,A 0.000,B 0.000,C 90.000,E1 77.521} C_DIS
LIN {X -0.052,Y -585.673,Z 1367.225,A 0.000,B 0.000,C 90.000,E1 76.464} C_DIS
